LIN {X 0,Y 517.01,Z 148.084,A -85,B 0,C 180,E1 -4953.117,E2 -4953.117} C_VEL
LIN {X 0,Y 516.998,Z 148.087,A -85,B 0,C 180,E1 -4956.243,E2 -4956.243} C_VEL
LIN {X 0,Y 516.949,Z 148.093,A -85,B 0,C 180,E1 -4959.389,E2 -4959.389} C_VEL
LIN {X 0,Y 516.95,Z 148.094,A -85,B 0,C 180,E1 -4961.808,E2 -4961.808} C_VEL
LIN {X 0,Y 516.941,Z 148.093,A -85,B 0,C 180,E1 -4965.147,E2 -4965.147} C_VEL
LIN {X 0,Y 516.922,Z 148.096,A -85,B 0,C 180,E1 -4968.222,E2 -4968.222} C_VEL
LIN {X 0,Y 516.909,Z 148.099,A -85,B 0,C 180,E1 -4970.702,E2 -4970.702} C_VEL
LIN {X 0,Y 516.909,Z 148.099,A -85,B 0,C 180,E1 -4974.072,E2 -4974.072} C_VEL
LIN {X 0,Y 516.923,Z 148.097,A -85,B 0,C 180,E1 -4976.658,E2 -4976.658} C_VEL
LIN {X 0,Y 516.909,Z 148.098,A -85,B 0,C 180,E1 -4979.524,E2 -4979.524} C_VEL
LIN {X 0,Y 516.895,Z 148.101,A -85,B 0,C 180,E1 -4982.544,E2 -4982.544} C_VEL
LIN {X 0,Y 516.863,Z 148.104,A -85,B 0,C 180,E1 -4985.33,E2 -4985.33} C_VEL
LIN {X 0,Y 516.878,Z 148.101,A -85,B 0,C 180,E1 -4987.943,E2 -4987.943} C_VEL
LIN {X 0,Y 516.883,Z 148.101,A -85,B 0,C 180,E1 -4990.742,E2 -4990.742} C_VEL
LIN {X 0,Y 516.882,Z 148.101,A -85,B 0,C 180,E1 -4992.832,E2 -4992.832} C_VEL
LIN {X 0,Y 516.921,Z 148.097,A -85,B 0,C 180,E1 -4995.01,E2 -4995.01} C_VEL
LIN {X 0,Y 516.911,Z 148.1,A -85,B 0,C 180,E1 -4998.399,E2 -4998.399} C_VEL
LIN {X 0,Y 516.88,Z 148.101,A -85,B 0,C 180,E1 -5001.285,E2 -5001.285} C_VEL
LIN {X 0,Y 516.885,Z 148.102,A -85,B 0,C 180,E1 -5004.221,E2 -5004.221} C_VEL
LIN {X 0,Y 516.88,Z 148.102,A -85,B 0,C 180,E1 -5007.053,E2 -5007.053} C_VEL
LIN {X 0,Y 516.891,Z 148.098,A -85,B 0,C 180,E1 -5009.797,E2 -5009.797} C_VEL
LIN {X 0,Y 516.925,Z 148.096,A -85,B 0,C 180,E1 -5012.468,E2 -5012.468} C_VEL
LIN {X 0,Y 516.908,Z 148.1,A -85,B 0,C 180,E1 -5015.072,E2 -5015.072} C_VEL
LIN {X 0,Y 516.886,Z 148.101,A -85,B 0,C 180,E1 -5018.463,E2 -5018.463} C_VEL
LIN {X 0,Y 516.901,Z 148.1,A -85,B 0,C 180,E1 -5020.955,E2 -5020.955} C_VEL
LIN {X 0,Y 516.906,Z 148.099,A -85,B 0,C 180,E1 -5023.41,E2 -5023.41} C_VEL
LIN {X 0,Y 516.893,Z 148.1,A -85,B 0,C 180,E1 -5025.834,E2 -5025.834} C_VEL
LIN {X 0,Y 516.967,Z 148.092,A -85,B 0,C 180,E1 -5028.234,E2 -5028.234} C_VEL
LIN {X 0,Y 516.96,Z 148.091,A -85,B 0,C 180,E1 -5031.4,E2 -5031.4} C_VEL
LIN {X 0,Y 517.012,Z 148.085,A -85,B 0,C 180,E1 -5033.757,E2 -5033.757} C_VEL
LIN {X 0,Y 517.086,Z 148.075,A -85,B 0,C 180,E1 -5037.664,E2 -5037.664} C_VEL
LIN {X 0,Y 517.094,Z 148.074,A -85,B 0,C 180,E1 -5040.779,E2 -5040.779} C_VEL
LIN {X 0,Y 517.013,Z 148.086,A -85,B 0,C 180,E1 -5043.117,E2 -5043.117} C_VEL
LIN {X 0,Y 516.996,Z 148.088,A -85,B 0,C 180,E1 -5046.244,E2 -5046.244} C_VEL
LIN {X 0,Y 516.945,Z 148.094,A -85,B 0,C 180,E1 -5049.39,E2 -5049.39} C_VEL
LIN {X 0,Y 516.955,Z 148.093,A -85,B 0,C 180,E1 -5051.807,E2 -5051.807} C_VEL
LIN {X 0,Y 516.946,Z 148.095,A -85,B 0,C 180,E1 -5055.146,E2 -5055.146} C_VEL
LIN {X 0,Y 516.927,Z 148.096,A -85,B 0,C 180,E1 -5058.222,E2 -5058.222} C_VEL
LIN {X 0,Y 516.915,Z 148.097,A -85,B 0,C 180,E1 -5060.702,E2 -5060.702} C_VEL
LIN {X 0,Y 516.904,Z 148.098,A -85,B 0,C 180,E1 -5064.073,E2 -5064.073} C_VEL
LIN {X 0,Y 516.928,Z 148.094,A -85,B 0,C 180,E1 -5066.658,E2 -5066.658} C_VEL
LIN {X 0,Y 516.913,Z 148.1,A -85,B 0,C 180,E1 -5069.524,E2 -5069.524} C_VEL
LIN {X 0,Y 516.897,Z 148.098,A -85,B 0,C 180,E1 -5072.543,E2 -5072.543} C_VEL
LIN {X 0,Y 516.868,Z 148.104,A -85,B 0,C 180,E1 -5075.33,E2 -5075.33} C_VEL
LIN {X 0,Y 516.882,Z 148.104,A -85,B 0,C 180,E1 -5077.943,E2 -5077.943} C_VEL
LIN {X 0,Y 516.885,Z 148.101,A -85,B 0,C 180,E1 -5080.742,E2 -5080.742} C_VEL
LIN {X 0,Y 516.885,Z 148.101,A -85,B 0,C 180,E1 -5082.832,E2 -5082.832} C_VEL
LIN {X 0,Y 516.926,Z 148.095,A -85,B 0,C 180,E1 -5085.01,E2 -5085.01} C_VEL
LIN {X 0,Y 516.916,Z 148.096,A -85,B 0,C 180,E1 -5088.399,E2 -5088.399} C_VEL
LIN {X 0,Y 516.917,Z 148.208,A -85,B 0,C 180,E1 -5091.168,E2 -5091.168} C_VEL
LIN {X 0,Y 518.075,Z 154.921,A -85,B 0,C 180,E1 -5093.836,E2 -5093.836} C_VEL
LIN {X 0,Y 518.083,Z 160.598,A -85,B 0,C 180,E1 -5095.842,E2 -5095.842} C_VEL
LIN {X 0,Y 517.83,Z 169.691,A -85,B 0,C 180,E1 -5098.953,E2 -5098.953} C_VEL
LIN {X 0,Y 517.591,Z 178.692,A -85,B 0,C 180,E1 -5101.957,E2 -5101.957} C_VEL
LIN {X 0,Y 517.294,Z 188.282,A -85,B 0,C 180,E1 -5105.092,E2 -5105.092} C_VEL
LIN {X 0,Y 517.074,Z 197.549,A -85,B 0,C 180,E1 -5108.051,E2 -5108.051} C_VEL
LIN {X 0,Y 516.881,Z 206.816,A -85,B 0,C 180,E1 -5110.954,E2 -5110.954} C_VEL
LIN {X 0,Y 516.684,Z 217.407,A -85,B 0,C 180,E1 -5114.214,E2 -5114.214} C_VEL
LIN {X 0,Y 516.588,Z 223.736,A -85,B 0,C 180,E1 -5116.095,E2 -5116.095} C_VEL
LIN {X 0,Y 518.516,Z 236.185,A -85,B 0,C 180,E1 -5116.429,E2 -5116.429} C_VEL
LIN {X 0,Y 518.261,Z 248.986,A -85,B 0,C 180,E1 -5116.871,E2 -5116.871} C_VEL
LIN {X 0,Y 517.942,Z 261.176,A -85,B 0,C 180,E1 -5117.461,E2 -5117.461} C_VEL
LIN {X 0,Y 517.617,Z 273.589,A -85,B 0,C 180,E1 -5118.249,E2 -5118.249} C_VEL
LIN {X 0,Y 517.327,Z 284.471,A -85,B 0,C 180,E1 -5119.135,E2 -5119.135} C_VEL
LIN {X 0,Y 517.045,Z 293.335,A -85,B 0,C 180,E1 -5120.02,E2 -5120.02} C_VEL
LIN {X 0,Y 516.814,Z 302.961,A -85,B 0,C 180,E1 -5121.2,E2 -5121.2} C_VEL
LIN {X 0,Y 516.563,Z 310.622,A -85,B 0,C 180,E1 -5122.377,E2 -5122.377} C_VEL
LIN {X 0,Y 516.427,Z 317.68,A -85,B 0,C 180,E1 -5123.75,E2 -5123.75} C_VEL
LIN {X 0,Y 516.313,Z 322.373,A -85,B 0,C 180,E1 -5124.924,E2 -5124.924} C_VEL
LIN {X 0,Y 516.355,Z 325.958,A -85,B 0,C 180,E1 -5126.098,E2 -5126.098} C_VEL
LIN {X 0,Y 516.282,Z 327.808,A -85,B 0,C 180,E1 -5126.879,E2 -5126.879} C_VEL
LIN {X 0,Y 516.261,Z 329.197,A -85,B 0,C 180,E1 -5127.66,E2 -5127.66} C_VEL
LIN {X 0,Y 516.16,Z 330.786,A -85,B 0,C 180,E1 -5129.22,E2 -5129.22} C_VEL
LIN {X 0,Y 516.154,Z 331,A -85,B 0,C 180,E1 -5130,E2 -5130} C_VEL
LIN {X 0,Y 516.192,Z 330.185,A -85,B 0,C 180,E1 -5131.561,E2 -5131.561} C_VEL
LIN {X 0,Y 516.262,Z 329.198,A -85,B 0,C 180,E1 -5132.341,E2 -5132.341} C_VEL
LIN {X 0,Y 516.283,Z 327.81,A -85,B 0,C 180,E1 -5133.121,E2 -5133.121} C_VEL
LIN {X 0,Y 516.344,Z 324.895,A -85,B 0,C 180,E1 -5134.293,E2 -5134.293} C_VEL
LIN {X 0,Y 516.406,Z 320.948,A -85,B 0,C 180,E1 -5135.467,E2 -5135.467} C_VEL
LIN {X 0,Y 516.487,Z 315.032,A -85,B 0,C 180,E1 -5136.808,E2 -5136.808} C_VEL
LIN {X 0,Y 516.641,Z 308.236,A -85,B 0,C 180,E1 -5138.015,E2 -5138.015} C_VEL
LIN {X 0,Y 516.868,Z 299.99,A -85,B 0,C 180,E1 -5139.194,E2 -5139.194} C_VEL
LIN {X 0,Y 517.081,Z 291.537,A -85,B 0,C 180,E1 -5140.177,E2 -5140.177} C_VEL
LIN {X 0,Y 517.435,Z 281.094,A -85,B 0,C 180,E1 -5141.16,E2 -5141.16} C_VEL
LIN {X 0,Y 517.698,Z 269.801,A -85,B 0,C 180,E1 -5142.014,E2 -5142.014} C_VEL
LIN {X 0,Y 517.987,Z 259.405,A -85,B 0,C 180,E1 -5142.638,E2 -5142.638} C_VEL
LIN {X 0,Y 518.27,Z 247.759,A -85,B 0,C 180,E1 -5143.179,E2 -5143.179} C_VEL
LIN {X 0,Y 518.431,Z 234.797,A -85,B 0,C 180,E1 -5143.611,E2 -5143.611} C_VEL
LIN {X 0,Y 516.571,Z 223.53,A -85,B 0,C 180,E1 -5143.924,E2 -5143.924} C_VEL
LIN {X 0,Y 516.712,Z 214.759,A -85,B 0,C 180,E1 -5146.597,E2 -5146.597} C_VEL
LIN {X 0,Y 516.907,Z 205.491,A -85,B 0,C 180,E1 -5149.458,E2 -5149.458} C_VEL
LIN {X 0,Y 517.1,Z 195.963,A -85,B 0,C 180,E1 -5152.451,E2 -5152.451} C_VEL
LIN {X 0,Y 517.324,Z 186.957,A -85,B 0,C 180,E1 -5155.337,E2 -5155.337} C_VEL
LIN {X 0,Y 517.604,Z 177.641,A -85,B 0,C 180,E1 -5158.374,E2 -5158.374} C_VEL
LIN {X 0,Y 517.843,Z 168.077,A -85,B 0,C 180,E1 -5161.55,E2 -5161.55} C_VEL
LIN {X 0,Y 518.14,Z 158.783,A -85,B 0,C 180,E1 -5164.728,E2 -5164.728} C_VEL
LIN {X 0,Y 518.062,Z 154.855,A -85,B 0,C 180,E1 -5166.166,E2 -5166.166} C_VEL
LIN {X 0,Y 516.901,Z 148.101,A -85,B 0,C 180,E1 -5168.893,E2 -5168.893} C_VEL
LIN {X 0,Y 516.918,Z 148.099,A -85,B 0,C 180,E1 -5171.775,E2 -5171.775} C_VEL
LIN {X 0,Y 516.927,Z 148.097,A -85,B 0,C 180,E1 -5175.01,E2 -5175.01} C_VEL
LIN {X 0,Y 516.919,Z 148.1,A -85,B 0,C 180,E1 -5178.399,E2 -5178.399} C_VEL
LIN {X 0,Y 516.886,Z 148.104,A -85,B 0,C 180,E1 -5181.284,E2 -5181.284} C_VEL
LIN {X 0,Y 516.876,Z 148.104,A -85,B 0,C 180,E1 -5184.22,E2 -5184.22} C_VEL
LIN {X 0,Y 516.901,Z 148.1,A -85,B 0,C 180,E1 -5187.053,E2 -5187.053} C_VEL
LIN {X 0,Y 516.897,Z 148.1,A -85,B 0,C 180,E1 -5189.796,E2 -5189.796} C_VEL
LIN {X 0,Y 516.933,Z 148.097,A -85,B 0,C 180,E1 -5192.467,E2 -5192.467} C_VEL
LIN {X 0,Y 516.914,Z 148.098,A -85,B 0,C 180,E1 -5195.072,E2 -5195.072} C_VEL
LIN {X 0,Y 516.891,Z 148.103,A -85,B 0,C 180,E1 -5198.462,E2 -5198.462} C_VEL
LIN {X 0,Y 516.905,Z 148.099,A -85,B 0,C 180,E1 -5200.955,E2 -5200.955} C_VEL
LIN {X 0,Y 516.91,Z 148.1,A -85,B 0,C 180,E1 -5203.41,E2 -5203.41} C_VEL
LIN {X 0,Y 516.9,Z 148.1,A -85,B 0,C 180,E1 -5205.833,E2 -5205.833} C_VEL
LIN {X 0,Y 516.971,Z 148.091,A -85,B 0,C 180,E1 -5208.233,E2 -5208.233} C_VEL
LIN {X 0,Y 516.973,Z 148.091,A -85,B 0,C 180,E1 -5211.399,E2 -5211.399} C_VEL
LIN {X 0,Y 517.016,Z 148.086,A -85,B 0,C 180,E1 -5213.757,E2 -5213.757} C_VEL
LIN {X 0,Y 517.089,Z 148.077,A -85,B 0,C 180,E1 -5217.663,E2 -5217.663} C_VEL
LIN {X 0,Y 517.098,Z 148.076,A -85,B 0,C 180,E1 -5220.778,E2 -5220.778} C_VEL
LIN {X 0,Y 517.016,Z 148.086,A -85,B 0,C 180,E1 -5223.117,E2 -5223.117} C_VEL
LIN {X 0,Y 517.013,Z 148.087,A -85,B 0,C 180,E1 -5226.243,E2 -5226.243} C_VEL
LIN {X 0,Y 516.957,Z 148.095,A -85,B 0,C 180,E1 -5228.6,E2 -5228.6} C_VEL
LIN {X 0,Y 516.756,Z 148.122,A -85,B 0,C 180,E1 -5230.976,E2 -5230.976} C_VEL
LIN {X 0,Y 516.707,Z 148.583,A -85,B 0,C 180,E1 -5231.772,E2 -5231.772} C_VEL
LIN {X 0,Y 516.661,Z 152.229,A -85,B 0,C 180,E1 -5235.028,E2 -5235.028} C_VEL
LIN {X 0,Y 516.555,Z 155.792,A -85,B 0,C 180,E1 -5238.235,E2 -5238.235} C_VEL
LIN {X 0,Y 516.478,Z 158.499,A -85,B 0,C 180,E1 -5240.719,E2 -5240.719} C_VEL
LIN {X 0,Y 516.437,Z 161.326,A -85,B 0,C 180,E1 -5243.244,E2 -5243.244} C_VEL
LIN {X 0,Y 516.458,Z 164.474,A -85,B 0,C 180,E1 -5246.086,E2 -5246.086} C_VEL
LIN {X 0,Y 516.396,Z 167.117,A -85,B 0,C 180,E1 -5248.446,E2 -5248.446} C_VEL
LIN {X 0,Y 516.39,Z 170.263,A -85,B 0,C 180,E1 -5251.228,E2 -5251.228} C_VEL
LIN {X 0,Y 518.487,Z 180.258,A -85,B 0,C 180,E1 -5251.542,E2 -5251.542} C_VEL
LIN {X 0,Y 518.265,Z 193.68,A -85,B 0,C 180,E1 -5252.043,E2 -5252.043} C_VEL
LIN {X 0,Y 518.01,Z 205.328,A -85,B 0,C 180,E1 -5252.635,E2 -5252.635} C_VEL
LIN {X 0,Y 517.692,Z 216.31,A -85,B 0,C 180,E1 -5253.354,E2 -5253.354} C_VEL
LIN {X 0,Y 517.434,Z 227.438,A -85,B 0,C 180,E1 -5254.28,E2 -5254.28} C_VEL
LIN {X 0,Y 517.201,Z 236.447,A -85,B 0,C 180,E1 -5255.204,E2 -5255.204} C_VEL
LIN {X 0,Y 516.915,Z 244.489,A -85,B 0,C 180,E1 -5256.204,E2 -5256.204} C_VEL
LIN {X 0,Y 516.718,Z 251.395,A -85,B 0,C 180,E1 -5257.247,E2 -5257.247} C_VEL
LIN {X 0,Y 516.568,Z 258.171,A -85,B 0,C 180,E1 -5258.521,E2 -5258.521} C_VEL
LIN {X 0,Y 516.422,Z 263.336,A -85,B 0,C 180,E1 -5259.763,E2 -5259.763} C_VEL
LIN {X 0,Y 516.356,Z 266.685,A -85,B 0,C 180,E1 -5260.791,E2 -5260.791} C_VEL
LIN {X 0,Y 516.322,Z 269.256,A -85,B 0,C 180,E1 -5261.833,E2 -5261.833} C_VEL
LIN {X 0,Y 516.274,Z 270.923,A -85,B 0,C 180,E1 -5262.775,E2 -5262.775} C_VEL
LIN {X 0,Y 515.597,Z 271.786,A -85,B 0,C 180,E1 -5263.42,E2 -5263.42} C_VEL
LIN {X 0,Y 512.694,Z 272.704,A -85,B 0,C 180,E1 -5264.472,E2 -5264.472} C_VEL
LIN {X 0,Y 510.257,Z 272.904,A -85,B 0,C 180,E1 -5265.322,E2 -5265.322} C_VEL
LIN {X 0,Y 509.229,Z 272.712,A -85,B 0,C 180,E1 -5265.979,E2 -5265.979} C_VEL
LIN {X 0,Y 509.157,Z 272.566,A -85,B 0,C 180,E1 -5266.201,E2 -5266.201} C_VEL
LIN {X 0,Y 509.204,Z 271.165,A -85,B 0,C 180,E1 -5267.445,E2 -5267.445} C_VEL
LIN {X 0,Y 509.249,Z 269.144,A -85,B 0,C 180,E1 -5268.514,E2 -5268.514} C_VEL
LIN {X 0,Y 509.305,Z 266.411,A -85,B 0,C 180,E1 -5269.566,E2 -5269.566} C_VEL
LIN {X 0,Y 509.438,Z 261.886,A -85,B 0,C 180,E1 -5270.865,E2 -5270.865} C_VEL
LIN {X 0,Y 509.574,Z 255.616,A -85,B 0,C 180,E1 -5272.237,E2 -5272.237} C_VEL
LIN {X 0,Y 509.751,Z 249.046,A -85,B 0,C 180,E1 -5273.374,E2 -5273.374} C_VEL
LIN {X 0,Y 509.996,Z 241.844,A -85,B 0,C 180,E1 -5274.394,E2 -5274.394} C_VEL
LIN {X 0,Y 510.322,Z 232.216,A -85,B 0,C 180,E1 -5275.503,E2 -5275.503} C_VEL
LIN {X 0,Y 510.604,Z 221.763,A -85,B 0,C 180,E1 -5276.476,E2 -5276.476} C_VEL
LIN {X 0,Y 510.87,Z 210.775,A -85,B 0,C 180,E1 -5277.294,E2 -5277.294} C_VEL
LIN {X 0,Y 511.199,Z 198.854,A -85,B 0,C 180,E1 -5277.984,E2 -5277.984} C_VEL
LIN {X 0,Y 511.527,Z 186.379,A -85,B 0,C 180,E1 -5278.527,E2 -5278.527} C_VEL
LIN {X 0,Y 511.357,Z 179.734,A -85,B 0,C 180,E1 -5278.758,E2 -5278.758} C_VEL
LIN {X 0,Y 509.272,Z 170.174,A -85,B 0,C 180,E1 -5279.07,E2 -5279.07} C_VEL
LIN {X 0,Y 509.287,Z 166.728,A -85,B 0,C 180,E1 -5282.027,E2 -5282.027} C_VEL
LIN {X 0,Y 509.343,Z 163.681,A -85,B 0,C 180,E1 -5284.675,E2 -5284.675} C_VEL
LIN {X 0,Y 509.318,Z 160.344,A -85,B 0,C 180,E1 -5287.595,E2 -5287.595} C_VEL
LIN {X 0,Y 509.349,Z 156.878,A -85,B 0,C 180,E1 -5290.661,E2 -5290.661} C_VEL
LIN {X 0,Y 509.419,Z 154.049,A -85,B 0,C 180,E1 -5293.159,E2 -5293.159} C_VEL
LIN {X 0,Y 509.504,Z 151.26,A -85,B 0,C 180,E1 -5295.624,E2 -5295.624} C_VEL
LIN {X 0,Y 509.523,Z 149.455,A -85,B 0,C 180,E1 -5297.25,E2 -5297.25} C_VEL
LIN {X 0,Y 509.655,Z 149.004,A -85,B 0,C 180,E1 -5298.255,E2 -5298.255} C_VEL
LIN {X 0,Y 509.894,Z 148.972,A -85,B 0,C 180,E1 -5301.279,E2 -5301.279} C_VEL
LIN {X 0,Y 509.941,Z 148.966,A -85,B 0,C 180,E1 -5303.67,E2 -5303.67} C_VEL
LIN {X 0,Y 509.952,Z 148.963,A -85,B 0,C 180,E1 -5306.84,E2 -5306.84} C_VEL
LIN {X 0,Y 510.06,Z 148.95,A -85,B 0,C 180,E1 -5309.21,E2 -5309.21} C_VEL
LIN {X 0,Y 510.053,Z 148.953,A -85,B 0,C 180,E1 -5312.369,E2 -5312.369} C_VEL
LIN {X 0,Y 509.976,Z 148.961,A -85,B 0,C 180,E1 -5315.536,E2 -5315.536} C_VEL
LIN {X 0,Y 509.948,Z 148.965,A -85,B 0,C 180,E1 -5317.921,E2 -5317.921} C_VEL
LIN {X 0,Y 509.91,Z 148.97,A -85,B 0,C 180,E1 -5321.125,E2 -5321.125} C_VEL
LIN {X 0,Y 509.861,Z 148.977,A -85,B 0,C 180,E1 -5324.366,E2 -5324.366} C_VEL
LIN {X 0,Y 509.899,Z 148.972,A -85,B 0,C 180,E1 -5327.652,E2 -5327.652} C_VEL
LIN {X 0,Y 509.883,Z 148.974,A -85,B 0,C 180,E1 -5330.402,E2 -5330.402} C_VEL
LIN {X 0,Y 509.834,Z 148.979,A -85,B 0,C 180,E1 -5333.563,E2 -5333.563} C_VEL
LIN {X 0,Y 509.909,Z 148.971,A -85,B 0,C 180,E1 -5336.379,E2 -5336.379} C_VEL
LIN {X 0,Y 509.874,Z 148.975,A -85,B 0,C 180,E1 -5338.844,E2 -5338.844} C_VEL
LIN {X 0,Y 509.819,Z 148.982,A -85,B 0,C 180,E1 -5341.59,E2 -5341.59} C_VEL
LIN {X 0,Y 509.844,Z 148.976,A -85,B 0,C 180,E1 -5344.414,E2 -5344.414} C_VEL
LIN {X 0,Y 509.814,Z 148.984,A -85,B 0,C 180,E1 -5347.341,E2 -5347.341} C_VEL
LIN {X 0,Y 509.836,Z 148.978,A -85,B 0,C 180,E1 -5350.382,E2 -5350.382} C_VEL
LIN {X 0,Y 509.822,Z 148.981,A -85,B 0,C 180,E1 -5353.063,E2 -5353.063} C_VEL
LIN {X 0,Y 509.829,Z 148.981,A -85,B 0,C 180,E1 -5355.793,E2 -5355.793} C_VEL
LIN {X 0,Y 509.853,Z 148.978,A -85,B 0,C 180,E1 -5358.575,E2 -5358.575} C_VEL
LIN {X 0,Y 509.85,Z 148.978,A -85,B 0,C 180,E1 -5361.787,E2 -5361.787} C_VEL
LIN {X 0,Y 509.841,Z 148.979,A -85,B 0,C 180,E1 -5364.623,E2 -5364.623} C_VEL
LIN {X 0,Y 509.859,Z 148.976,A -85,B 0,C 180,E1 -5367.481,E2 -5367.481} C_VEL
LIN {X 0,Y 509.857,Z 148.977,A -85,B 0,C 180,E1 -5370.274,E2 -5370.274} C_VEL
LIN {X 0,Y 509.883,Z 148.974,A -85,B 0,C 180,E1 -5372.945,E2 -5372.945} C_VEL
LIN {X 0,Y 509.864,Z 148.974,A -85,B 0,C 180,E1 -5375.574,E2 -5375.574} C_VEL
LIN {X 0,Y 509.851,Z 148.977,A -85,B 0,C 180,E1 -5378.999,E2 -5378.999} C_VEL
LIN {X 0,Y 509.862,Z 148.976,A -85,B 0,C 180,E1 -5381.517,E2 -5381.517} C_VEL
LIN {X 0,Y 509.911,Z 148.971,A -85,B 0,C 180,E1 -5384.819,E2 -5384.819} C_VEL
LIN {X 0,Y 509.902,Z 148.971,A -85,B 0,C 180,E1 -5388.124,E2 -5388.124} C_VEL
LIN {X 0,Y 509.908,Z 148.969,A -85,B 0,C 180,E1 -5391.28,E2 -5391.28} C_VEL
LIN {X 0,Y 509.981,Z 148.961,A -85,B 0,C 180,E1 -5393.671,E2 -5393.671} C_VEL
LIN {X 0,Y 510.057,Z 148.951,A -85,B 0,C 180,E1 -5397.631,E2 -5397.631} C_VEL
LIN {X 0,Y 510.065,Z 148.95,A -85,B 0,C 180,E1 -5400.79,E2 -5400.79} C_VEL
LIN {X 0,Y 509.955,Z 148.965,A -85,B 0,C 180,E1 -5403.161,E2 -5403.161} C_VEL
LIN {X 0,Y 509.944,Z 148.967,A -85,B 0,C 180,E1 -5406.33,E2 -5406.33} C_VEL
LIN {X 0,Y 509.906,Z 148.971,A -85,B 0,C 180,E1 -5408.721,E2 -5408.721} C_VEL
LIN {X 0,Y 509.907,Z 148.97,A -85,B 0,C 180,E1 -5411.932,E2 -5411.932} C_VEL
LIN {X 0,Y 509.897,Z 148.973,A -85,B 0,C 180,E1 -5415.242,E2 -5415.242} C_VEL
LIN {X 0,Y 509.885,Z 148.973,A -85,B 0,C 180,E1 -5417.999,E2 -5417.999} C_VEL
LIN {X 0,Y 509.853,Z 148.978,A -85,B 0,C 180,E1 -5421.002,E2 -5421.002} C_VEL
LIN {X 0,Y 509.866,Z 148.976,A -85,B 0,C 180,E1 -5424.427,E2 -5424.427} C_VEL
LIN {X 0,Y 509.887,Z 148.974,A -85,B 0,C 180,E1 -5427.056,E2 -5427.056} C_VEL
LIN {X 0,Y 509.86,Z 148.976,A -85,B 0,C 180,E1 -5429.751,E2 -5429.751} C_VEL
LIN {X 0,Y 509.869,Z 148.974,A -85,B 0,C 180,E1 -5432.773,E2 -5432.773} C_VEL
LIN {X 0,Y 509.828,Z 148.981,A -85,B 0,C 180,E1 -5435.579,E2 -5435.579} C_VEL
LIN {X 0,Y 509.852,Z 148.977,A -85,B 0,C 180,E1 -5438.338,E2 -5438.338} C_VEL
LIN {X 0,Y 509.858,Z 148.978,A -85,B 0,C 180,E1 -5441.426,E2 -5441.426} C_VEL
LIN {X 0,Y 509.859,Z 148.973,A -85,B 0,C 180,E1 -5444.668,E2 -5444.668} C_VEL
LIN {X 0,Y 509.858,Z 148.975,A -85,B 0,C 180,E1 -5448.104,E2 -5448.104} C_VEL
LIN {X 0,Y 509.876,Z 149.163,A -85,B 0,C 180,E1 -5450.905,E2 -5450.905} C_VEL
LIN {X 0,Y 511.095,Z 156.154,A -85,B 0,C 180,E1 -5453.752,E2 -5453.752} C_VEL
LIN {X 0,Y 511.114,Z 161.509,A -85,B 0,C 180,E1 -5455.683,E2 -5455.683} C_VEL
LIN {X 0,Y 510.88,Z 169.695,A -85,B 0,C 180,E1 -5458.53,E2 -5458.53} C_VEL
LIN {X 0,Y 510.591,Z 179.233,A -85,B 0,C 180,E1 -5461.755,E2 -5461.755} C_VEL
LIN {X 0,Y 510.302,Z 188.282,A -85,B 0,C 180,E1 -5464.727,E2 -5464.727} C_VEL
LIN {X 0,Y 510.081,Z 197.673,A -85,B 0,C 180,E1 -5467.774,E2 -5467.774} C_VEL
LIN {X 0,Y 509.859,Z 206.816,A -85,B 0,C 180,E1 -5470.681,E2 -5470.681} C_VEL
LIN {X 0,Y 509.647,Z 217.407,A -85,B 0,C 180,E1 -5473.99,E2 -5473.99} C_VEL
LIN {X 0,Y 509.54,Z 223.736,A -85,B 0,C 180,E1 -5475.899,E2 -5475.899} C_VEL
LIN {X 0,Y 511.617,Z 236.642,A -85,B 0,C 180,E1 -5476.255,E2 -5476.255} C_VEL
LIN {X 0,Y 511.36,Z 248.985,A -85,B 0,C 180,E1 -5476.691,E2 -5476.691} C_VEL
LIN {X 0,Y 510.995,Z 261.176,A -85,B 0,C 180,E1 -5477.288,E2 -5477.288} C_VEL
LIN {X 0,Y 510.742,Z 271.848,A -85,B 0,C 180,E1 -5477.964,E2 -5477.964} C_VEL
LIN {X 0,Y 510.416,Z 282.264,A -85,B 0,C 180,E1 -5478.785,E2 -5478.785} C_VEL
LIN {X 0,Y 510.07,Z 291.54,A -85,B 0,C 180,E1 -5479.682,E2 -5479.682} C_VEL
LIN {X 0,Y 509.846,Z 299.992,A -85,B 0,C 180,E1 -5480.679,E2 -5480.679} C_VEL
LIN {X 0,Y 509.585,Z 308.237,A -85,B 0,C 180,E1 -5481.873,E2 -5481.873} C_VEL
LIN {X 0,Y 509.419,Z 314.878,A -85,B 0,C 180,E1 -5483.067,E2 -5483.067} C_VEL
LIN {X 0,Y 509.344,Z 320.95,A -85,B 0,C 180,E1 -5484.457,E2 -5484.457} C_VEL
LIN {X 0,Y 509.234,Z 324.895,A -85,B 0,C 180,E1 -5485.647,E2 -5485.647} C_VEL
LIN {X 0,Y 509.201,Z 327.808,A -85,B 0,C 180,E1 -5486.835,E2 -5486.835} C_VEL
LIN {X 0,Y 509.162,Z 329.196,A -85,B 0,C 180,E1 -5487.627,E2 -5487.627} C_VEL
LIN {X 0,Y 509.073,Z 330.786,A -85,B 0,C 180,E1 -5489.209,E2 -5489.209} C_VEL
LIN {X 0,Y 509.065,Z 331,A -85,B 0,C 180,E1 -5490,E2 -5490} C_VEL
LIN {X 0,Y 509.113,Z 330.185,A -85,B 0,C 180,E1 -5491.582,E2 -5491.582} C_VEL
LIN {X 0,Y 509.162,Z 329.198,A -85,B 0,C 180,E1 -5492.373,E2 -5492.373} C_VEL
LIN {X 0,Y 509.201,Z 327.81,A -85,B 0,C 180,E1 -5493.165,E2 -5493.165} C_VEL
LIN {X 0,Y 509.234,Z 324.895,A -85,B 0,C 180,E1 -5494.353,E2 -5494.353} C_VEL
LIN {X 0,Y 509.345,Z 320.948,A -85,B 0,C 180,E1 -5495.543,E2 -5495.543} C_VEL
LIN {X 0,Y 509.411,Z 315.281,A -85,B 0,C 180,E1 -5496.854,E2 -5496.854} C_VEL
LIN {X 0,Y 509.586,Z 308.235,A -85,B 0,C 180,E1 -5498.127,E2 -5498.127} C_VEL
LIN {X 0,Y 509.847,Z 299.99,A -85,B 0,C 180,E1 -5499.321,E2 -5499.321} C_VEL
LIN {X 0,Y 510.07,Z 291.537,A -85,B 0,C 180,E1 -5500.319,E2 -5500.319} C_VEL
LIN {X 0,Y 510.452,Z 281.093,A -85,B 0,C 180,E1 -5501.315,E2 -5501.315} C_VEL
LIN {X 0,Y 510.731,Z 270.53,A -85,B 0,C 180,E1 -5502.129,E2 -5502.129} C_VEL
LIN {X 0,Y 511.044,Z 259.404,A -85,B 0,C 180,E1 -5502.812,E2 -5502.812} C_VEL
LIN {X 0,Y 511.376,Z 247.759,A -85,B 0,C 180,E1 -5503.36,E2 -5503.36} C_VEL
LIN {X 0,Y 511.433,Z 235.254,A -85,B 0,C 180,E1 -5503.788,E2 -5503.788} C_VEL
LIN {X 0,Y 509.531,Z 223.53,A -85,B 0,C 180,E1 -5504.121,E2 -5504.121} C_VEL
LIN {X 0,Y 509.718,Z 213.435,A -85,B 0,C 180,E1 -5507.244,E2 -5507.244} C_VEL
LIN {X 0,Y 509.925,Z 204.167,A -85,B 0,C 180,E1 -5510.155,E2 -5510.155} C_VEL
LIN {X 0,Y 510.123,Z 194.9,A -85,B 0,C 180,E1 -5513.12,E2 -5513.12} C_VEL
LIN {X 0,Y 510.372,Z 185.572,A -85,B 0,C 180,E1 -5516.146,E2 -5516.146} C_VEL
LIN {X 0,Y 510.608,Z 177.504,A -85,B 0,C 180,E1 -5518.799,E2 -5518.799} C_VEL
LIN {X 0,Y 510.855,Z 169.425,A -85,B 0,C 180,E1 -5521.519,E2 -5521.519} C_VEL
LIN {X 0,Y 511.178,Z 159.957,A -85,B 0,C 180,E1 -5524.793,E2 -5524.793} C_VEL
LIN {X 0,Y 510.964,Z 155.063,A -85,B 0,C 180,E1 -5526.65,E2 -5526.65} C_VEL
LIN {X 0,Y 509.852,Z 148.979,A -85,B 0,C 180,E1 -5529.225,E2 -5529.225} C_VEL
LIN {X 0,Y 509.862,Z 148.977,A -85,B 0,C 180,E1 -5531.897,E2 -5531.897} C_VEL
LIN {X 0,Y 509.861,Z 148.979,A -85,B 0,C 180,E1 -5535.332,E2 -5535.332} C_VEL
LIN {X 0,Y 509.861,Z 148.979,A -85,B 0,C 180,E1 -5538.575,E2 -5538.575} C_VEL
LIN {X 0,Y 509.856,Z 148.979,A -85,B 0,C 180,E1 -5541.786,E2 -5541.786} C_VEL
LIN {X 0,Y 509.835,Z 148.981,A -85,B 0,C 180,E1 -5544.622,E2 -5544.622} C_VEL
LIN {X 0,Y 509.868,Z 148.976,A -85,B 0,C 180,E1 -5547.481,E2 -5547.481} C_VEL
LIN {X 0,Y 509.863,Z 148.978,A -85,B 0,C 180,E1 -5550.274,E2 -5550.274} C_VEL
LIN {X 0,Y 509.89,Z 148.972,A -85,B 0,C 180,E1 -5552.944,E2 -5552.944} C_VEL
LIN {X 0,Y 509.869,Z 148.976,A -85,B 0,C 180,E1 -5555.574,E2 -5555.574} C_VEL
LIN {X 0,Y 509.855,Z 148.977,A -85,B 0,C 180,E1 -5558.998,E2 -5558.998} C_VEL
LIN {X 0,Y 509.866,Z 148.976,A -85,B 0,C 180,E1 -5561.516,E2 -5561.516} C_VEL
LIN {X 0,Y 509.916,Z 148.97,A -85,B 0,C 180,E1 -5564.819,E2 -5564.819} C_VEL
LIN {X 0,Y 509.906,Z 148.971,A -85,B 0,C 180,E1 -5568.124,E2 -5568.124} C_VEL
LIN {X 0,Y 509.92,Z 148.97,A -85,B 0,C 180,E1 -5571.279,E2 -5571.279} C_VEL
LIN {X 0,Y 509.984,Z 148.963,A -85,B 0,C 180,E1 -5573.67,E2 -5573.67} C_VEL
LIN {X 0,Y 510.06,Z 148.953,A -85,B 0,C 180,E1 -5577.631,E2 -5577.631} C_VEL
LIN {X 0,Y 510.068,Z 148.951,A -85,B 0,C 180,E1 -5580.789,E2 -5580.789} C_VEL
LIN {X 0,Y 509.958,Z 148.965,A -85,B 0,C 180,E1 -5583.16,E2 -5583.16} C_VEL
LIN {X 0,Y 509.982,Z 148.963,A -85,B 0,C 180,E1 -5586.329,E2 -5586.329} C_VEL
LIN {X 0,Y 509.899,Z 148.974,A -85,B 0,C 180,E1 -5588.72,E2 -5588.72} C_VEL
LIN {X 0,Y 509.695,Z 149.001,A -85,B 0,C 180,E1 -5591.13,E2 -5591.13} C_VEL
LIN {X 0,Y 509.635,Z 149.582,A -85,B 0,C 180,E1 -5591.938,E2 -5591.938} C_VEL
LIN {X 0,Y 509.589,Z 153.184,A -85,B 0,C 180,E1 -5595.191,E2 -5595.191} C_VEL
LIN {X 0,Y 509.479,Z 156.8,A -85,B 0,C 180,E1 -5598.498,E2 -5598.498} C_VEL
LIN {X 0,Y 509.401,Z 159.606,A -85,B 0,C 180,E1 -5601.021,E2 -5601.021} C_VEL
LIN {X 0,Y 509.348,Z 162.415,A -85,B 0,C 180,E1 -5603.587,E2 -5603.587} C_VEL
LIN {X 0,Y 509.406,Z 165.381,A -85,B 0,C 180,E1 -5606.263,E2 -5606.263} C_VEL
LIN {X 0,Y 509.323,Z 168.295,A -85,B 0,C 180,E1 -5608.878,E2 -5608.878} C_VEL
LIN {X 0,Y 509.335,Z 170.743,A -85,B 0,C 180,E1 -5611.037,E2 -5611.037} C_VEL
LIN {X 0,Y 511.622,Z 181.465,A -85,B 0,C 180,E1 -5611.386,E2 -5611.386} C_VEL
LIN {X 0,Y 511.352,Z 194.845,A -85,B 0,C 180,E1 -5611.901,E2 -5611.901} C_VEL
LIN {X 0,Y 511.06,Z 206.685,A -85,B 0,C 180,E1 -5612.521,E2 -5612.521} C_VEL
LIN {X 0,Y 510.734,Z 217.646,A -85,B 0,C 180,E1 -5613.266,E2 -5613.266} C_VEL
LIN {X 0,Y 510.434,Z 228.789,A -85,B 0,C 180,E1 -5614.221,E2 -5614.221} C_VEL
LIN {X 0,Y 510.153,Z 238.29,A -85,B 0,C 180,E1 -5615.231,E2 -5615.231} C_VEL
LIN {X 0,Y 509.838,Z 246.793,A -85,B 0,C 180,E1 -5616.351,E2 -5616.351} C_VEL
LIN {X 0,Y 509.639,Z 254.187,A -85,B 0,C 180,E1 -5617.558,E2 -5617.558} C_VEL
LIN {X 0,Y 509.46,Z 260.61,A -85,B 0,C 180,E1 -5618.878,E2 -5618.878} C_VEL
LIN {X 0,Y 509.355,Z 264.546,A -85,B 0,C 180,E1 -5619.91,E2 -5619.91} C_VEL
LIN {X 0,Y 509.266,Z 267.894,A -85,B 0,C 180,E1 -5621.025,E2 -5621.025} C_VEL
LIN {X 0,Y 509.256,Z 269.76,A -85,B 0,C 180,E1 -5621.821,E2 -5621.821} C_VEL
LIN {X 0,Y 509.196,Z 271.693,A -85,B 0,C 180,E1 -5622.986,E2 -5622.986} C_VEL
LIN {X 0,Y 509.15,Z 272.744,A -85,B 0,C 180,E1 -5624.128,E2 -5624.128} C_VEL
LIN {X 0,Y 509.147,Z 272.987,A -85,B 0,C 180,E1 -5625.253,E2 -5625.253} C_VEL
LIN {X 0,Y 509.157,Z 272.566,A -85,B 0,C 180,E1 -5626.201,E2 -5626.201} C_VEL
LIN {X 0,Y 508.521,Z 272.042,A -85,B 0,C 180,E1 -5626.861,E2 -5626.861} C_VEL
LIN {X 0,Y 505.692,Z 270.711,A -85,B 0,C 180,E1 -5627.926,E2 -5627.926} C_VEL
LIN {X 0,Y 503.304,Z 269.091,A -85,B 0,C 180,E1 -5628.771,E2 -5628.771} C_VEL
LIN {X 0,Y 502.299,Z 267.463,A -85,B 0,C 180,E1 -5629.412,E2 -5629.412} C_VEL
LIN {X 0,Y 502.23,Z 266.832,A -85,B 0,C 180,E1 -5629.626,E2 -5629.626} C_VEL
LIN {X 0,Y 502.383,Z 262.138,A -85,B 0,C 180,E1 -5630.985,E2 -5630.985} C_VEL
LIN {X 0,Y 502.51,Z 256.492,A -85,B 0,C 180,E1 -5632.242,E2 -5632.242} C_VEL
LIN {X 0,Y 502.755,Z 249.052,A -85,B 0,C 180,E1 -5633.551,E2 -5633.551} C_VEL
LIN {X 0,Y 503.058,Z 240.93,A -85,B 0,C 180,E1 -5634.687,E2 -5634.687} C_VEL
LIN {X 0,Y 503.336,Z 232.635,A -85,B 0,C 180,E1 -5635.644,E2 -5635.644} C_VEL
LIN {X 0,Y 503.643,Z 222.563,A -85,B 0,C 180,E1 -5636.597,E2 -5636.597} C_VEL
LIN {X 0,Y 503.916,Z 212.012,A -85,B 0,C 180,E1 -5637.405,E2 -5637.405} C_VEL
LIN {X 0,Y 504.277,Z 200.675,A -85,B 0,C 180,E1 -5638.087,E2 -5638.087} C_VEL
LIN {X 0,Y 504.63,Z 187.628,A -85,B 0,C 180,E1 -5638.677,E2 -5638.677} C_VEL
LIN {X 0,Y 504.575,Z 181.35,A -85,B 0,C 180,E1 -5638.902,E2 -5638.902} C_VEL
LIN {X 0,Y 502.172,Z 170.533,A -85,B 0,C 180,E1 -5639.281,E2 -5639.281} C_VEL
LIN {X 0,Y 502.206,Z 166.815,A -85,B 0,C 180,E1 -5642.496,E2 -5642.496} C_VEL
LIN {X 0,Y 502.237,Z 163.737,A -85,B 0,C 180,E1 -5645.178,E2 -5645.178} C_VEL
LIN {X 0,Y 502.27,Z 160.751,A -85,B 0,C 180,E1 -5647.802,E2 -5647.802} C_VEL
LIN {X 0,Y 502.281,Z 157.844,A -85,B 0,C 180,E1 -5650.378,E2 -5650.378} C_VEL
LIN {X 0,Y 502.363,Z 154.991,A -85,B 0,C 180,E1 -5652.915,E2 -5652.915} C_VEL
LIN {X 0,Y 502.439,Z 152.19,A -85,B 0,C 180,E1 -5655.417,E2 -5655.417} C_VEL
LIN {X 0,Y 502.447,Z 150.358,A -85,B 0,C 180,E1 -5657.067,E2 -5657.067} C_VEL
LIN {X 0,Y 502.597,Z 149.883,A -85,B 0,C 180,E1 -5658.189,E2 -5658.189} C_VEL
LIN {X 0,Y 502.848,Z 149.849,A -85,B 0,C 180,E1 -5661.156,E2 -5661.156} C_VEL
LIN {X 0,Y 502.893,Z 149.843,A -85,B 0,C 180,E1 -5663.581,E2 -5663.581} C_VEL
LIN {X 0,Y 502.895,Z 149.842,A -85,B 0,C 180,E1 -5666.795,E2 -5666.795} C_VEL
LIN {X 0,Y 503.031,Z 149.826,A -85,B 0,C 180,E1 -5669.199,E2 -5669.199} C_VEL
LIN {X 0,Y 502.901,Z 149.843,A -85,B 0,C 180,E1 -5671.601,E2 -5671.601} C_VEL
LIN {X 0,Y 502.895,Z 149.842,A -85,B 0,C 180,E1 -5673.204,E2 -5673.204} C_VEL
LIN {X 0,Y 502.902,Z 149.842,A -85,B 0,C 180,E1 -5676.419,E2 -5676.419} C_VEL
LIN {X 0,Y 502.87,Z 149.846,A -85,B 0,C 180,E1 -5678.843,E2 -5678.843} C_VEL
LIN {X 0,Y 502.843,Z 149.851,A -85,B 0,C 180,E1 -5682.102,E2 -5682.102} C_VEL
LIN {X 0,Y 502.845,Z 149.85,A -85,B 0,C 180,E1 -5685.4,E2 -5685.4} C_VEL
LIN {X 0,Y 502.843,Z 149.851,A -85,B 0,C 180,E1 -5688.122,E2 -5688.122} C_VEL
LIN {X 0,Y 502.825,Z 149.853,A -85,B 0,C 180,E1 -5690.536,E2 -5690.536} C_VEL
LIN {X 0,Y 502.794,Z 149.858,A -85,B 0,C 180,E1 -5693.04,E2 -5693.04} C_VEL
LIN {X 0,Y 502.837,Z 149.851,A -85,B 0,C 180,E1 -5695.676,E2 -5695.676} C_VEL
LIN {X 0,Y 502.837,Z 149.849,A -85,B 0,C 180,E1 -5698.373,E2 -5698.373} C_VEL
LIN {X 0,Y 502.791,Z 149.858,A -85,B 0,C 180,E1 -5701.499,E2 -5701.499} C_VEL
LIN {X 0,Y 502.801,Z 149.855,A -85,B 0,C 180,E1 -5703.994,E2 -5703.994} C_VEL
LIN {X 0,Y 502.775,Z 149.86,A -85,B 0,C 180,E1 -5707.178,E2 -5707.178} C_VEL
LIN {X 0,Y 502.786,Z 149.857,A -85,B 0,C 180,E1 -5710.015,E2 -5710.015} C_VEL
LIN {X 0,Y 502.8,Z 149.856,A -85,B 0,C 180,E1 -5712.2,E2 -5712.2} C_VEL
LIN {X 0,Y 502.799,Z 149.856,A -85,B 0,C 180,E1 -5715.469,E2 -5715.469} C_VEL
LIN {X 0,Y 502.817,Z 149.853,A -85,B 0,C 180,E1 -5718.934,E2 -5718.934} C_VEL
LIN {X 0,Y 502.792,Z 149.857,A -85,B 0,C 180,E1 -5722.047,E2 -5722.047} C_VEL
LIN {X 0,Y 502.802,Z 149.855,A -85,B 0,C 180,E1 -5725.035,E2 -5725.035} C_VEL
LIN {X 0,Y 502.781,Z 149.858,A -85,B 0,C 180,E1 -5727.916,E2 -5727.916} C_VEL
LIN {X 0,Y 502.822,Z 149.853,A -85,B 0,C 180,E1 -5730.713,E2 -5730.713} C_VEL
LIN {X 0,Y 502.862,Z 149.847,A -85,B 0,C 180,E1 -5733.44,E2 -5733.44} C_VEL
LIN {X 0,Y 502.785,Z 149.857,A -85,B 0,C 180,E1 -5736.086,E2 -5736.086} C_VEL
LIN {X 0,Y 502.784,Z 149.86,A -85,B 0,C 180,E1 -5738.689,E2 -5738.689} C_VEL
LIN {X 0,Y 502.827,Z 149.852,A -85,B 0,C 180,E1 -5741.249,E2 -5741.249} C_VEL
LIN {X 0,Y 502.849,Z 149.851,A -85,B 0,C 180,E1 -5744.601,E2 -5744.601} C_VEL
LIN {X 0,Y 502.877,Z 149.846,A -85,B 0,C 180,E1 -5748.04,E2 -5748.04} C_VEL
LIN {X 0,Y 502.869,Z 149.846,A -85,B 0,C 180,E1 -5751.157,E2 -5751.157} C_VEL
LIN {X 0,Y 502.93,Z 149.84,A -85,B 0,C 180,E1 -5753.582,E2 -5753.582} C_VEL
LIN {X 0,Y 502.9,Z 149.844,A -85,B 0,C 180,E1 -5756.796,E2 -5756.796} C_VEL
LIN {X 0,Y 503.036,Z 149.826,A -85,B 0,C 180,E1 -5759.2,E2 -5759.2} C_VEL
LIN {X 0,Y 502.901,Z 149.843,A -85,B 0,C 180,E1 -5761.602,E2 -5761.602} C_VEL
LIN {X 0,Y 502.899,Z 149.844,A -85,B 0,C 180,E1 -5763.205,E2 -5763.205} C_VEL
LIN {X 0,Y 502.893,Z 149.846,A -85,B 0,C 180,E1 -5766.42,E2 -5766.42} C_VEL
LIN {X 0,Y 502.866,Z 149.848,A -85,B 0,C 180,E1 -5768.844,E2 -5768.844} C_VEL
LIN {X 0,Y 502.849,Z 149.85,A -85,B 0,C 180,E1 -5772.102,E2 -5772.102} C_VEL
LIN {X 0,Y 502.851,Z 149.85,A -85,B 0,C 180,E1 -5775.4,E2 -5775.4} C_VEL
LIN {X 0,Y 502.843,Z 149.85,A -85,B 0,C 180,E1 -5778.121,E2 -5778.121} C_VEL
LIN {X 0,Y 502.832,Z 149.85,A -85,B 0,C 180,E1 -5780.536,E2 -5780.536} C_VEL
LIN {X 0,Y 502.793,Z 149.856,A -85,B 0,C 180,E1 -5783.041,E2 -5783.041} C_VEL
LIN {X 0,Y 502.843,Z 149.852,A -85,B 0,C 180,E1 -5785.676,E2 -5785.676} C_VEL
LIN {X 0,Y 502.842,Z 149.851,A -85,B 0,C 180,E1 -5788.373,E2 -5788.373} C_VEL
LIN {X 0,Y 502.795,Z 149.857,A -85,B 0,C 180,E1 -5791.499,E2 -5791.499} C_VEL
LIN {X 0,Y 502.791,Z 149.857,A -85,B 0,C 180,E1 -5793.995,E2 -5793.995} C_VEL
LIN {X 0,Y 502.78,Z 149.858,A -85,B 0,C 180,E1 -5797.178,E2 -5797.178} C_VEL
LIN {X 0,Y 502.79,Z 149.857,A -85,B 0,C 180,E1 -5800.015,E2 -5800.015} C_VEL
LIN {X 0,Y 502.805,Z 149.853,A -85,B 0,C 180,E1 -5802.199,E2 -5802.199} C_VEL
LIN {X 0,Y 502.803,Z 149.853,A -85,B 0,C 180,E1 -5805.468,E2 -5805.468} C_VEL
LIN {X 0,Y 502.822,Z 149.853,A -85,B 0,C 180,E1 -5808.934,E2 -5808.934} C_VEL
LIN {X 0,Y 502.808,Z 149.948,A -85,B 0,C 180,E1 -5810.572,E2 -5810.572} C_VEL
LIN {X 0,Y 503.957,Z 156.175,A -85,B 0,C 180,E1 -5813.154,E2 -5813.154} C_VEL
LIN {X 0,Y 504.253,Z 160.027,A -85,B 0,C 180,E1 -5814.662,E2 -5814.662} C_VEL
LIN {X 0,Y 503.958,Z 168.083,A -85,B 0,C 180,E1 -5817.527,E2 -5817.527} C_VEL
LIN {X 0,Y 503.683,Z 176.159,A -85,B 0,C 180,E1 -5820.323,E2 -5820.323} C_VEL
LIN {X 0,Y 503.442,Z 183.972,A -85,B 0,C 180,E1 -5822.988,E2 -5822.988} C_VEL
LIN {X 0,Y 503.213,Z 192.215,A -85,B 0,C 180,E1 -5825.669,E2 -5825.669} C_VEL
LIN {X 0,Y 502.968,Z 201.521,A -85,B 0,C 180,E1 -5828.697,E2 -5828.697} C_VEL
LIN {X 0,Y 502.716,Z 211.598,A -85,B 0,C 180,E1 -5831.924,E2 -5831.924} C_VEL
LIN {X 0,Y 502.514,Z 221.694,A -85,B 0,C 180,E1 -5835.104,E2 -5835.104} C_VEL
LIN {X 0,Y 502.486,Z 223.582,A -85,B 0,C 180,E1 -5835.693,E2 -5835.693} C_VEL
LIN {X 0,Y 504.672,Z 237.098,A -85,B 0,C 180,E1 -5836.075,E2 -5836.075} C_VEL
LIN {X 0,Y 504.403,Z 250.114,A -85,B 0,C 180,E1 -5836.555,E2 -5836.555} C_VEL
LIN {X 0,Y 504.035,Z 262.527,A -85,B 0,C 180,E1 -5837.188,E2 -5837.188} C_VEL
LIN {X 0,Y 503.696,Z 273.59,A -85,B 0,C 180,E1 -5837.919,E2 -5837.919} C_VEL
LIN {X 0,Y 503.371,Z 284.47,A -85,B 0,C 180,E1 -5838.83,E2 -5838.83} C_VEL
LIN {X 0,Y 503.023,Z 293.335,A -85,B 0,C 180,E1 -5839.739,E2 -5839.739} C_VEL
LIN {X 0,Y 502.705,Z 302.961,A -85,B 0,C 180,E1 -5840.951,E2 -5840.951} C_VEL
LIN {X 0,Y 502.471,Z 310.622,A -85,B 0,C 180,E1 -5842.162,E2 -5842.162} C_VEL
LIN {X 0,Y 502.256,Z 317.68,A -85,B 0,C 180,E1 -5843.573,E2 -5843.573} C_VEL
LIN {X 0,Y 502.186,Z 322.373,A -85,B 0,C 180,E1 -5844.781,E2 -5844.781} C_VEL
LIN {X 0,Y 502.152,Z 325.958,A -85,B 0,C 180,E1 -5845.987,E2 -5845.987} C_VEL
LIN {X 0,Y 502.121,Z 327.808,A -85,B 0,C 180,E1 -5846.791,E2 -5846.791} C_VEL
LIN {X 0,Y 502.066,Z 329.195,A -85,B 0,C 180,E1 -5847.593,E2 -5847.593} C_VEL
LIN {X 0,Y 501.99,Z 330.786,A -85,B 0,C 180,E1 -5849.198,E2 -5849.198} C_VEL
LIN {X 0,Y 501.98,Z 331,A -85,B 0,C 180,E1 -5850,E2 -5850} C_VEL
LIN {X 0,Y 502.036,Z 330.185,A -85,B 0,C 180,E1 -5851.605,E2 -5851.605} C_VEL
LIN {X 0,Y 502.066,Z 329.197,A -85,B 0,C 180,E1 -5852.407,E2 -5852.407} C_VEL
LIN {X 0,Y 502.121,Z 327.81,A -85,B 0,C 180,E1 -5853.21,E2 -5853.21} C_VEL
LIN {X 0,Y 502.128,Z 324.895,A -85,B 0,C 180,E1 -5854.415,E2 -5854.415} C_VEL
LIN {X 0,Y 502.26,Z 320.948,A -85,B 0,C 180,E1 -5855.621,E2 -5855.621} C_VEL
LIN {X 0,Y 502.336,Z 314.976,A -85,B 0,C 180,E1 -5857.012,E2 -5857.012} C_VEL
LIN {X 0,Y 502.543,Z 308.235,A -85,B 0,C 180,E1 -5858.242,E2 -5858.242} C_VEL
LIN {X 0,Y 502.812,Z 299.99,A -85,B 0,C 180,E1 -5859.453,E2 -5859.453} C_VEL
LIN {X 0,Y 503.064,Z 291.538,A -85,B 0,C 180,E1 -5860.464,E2 -5860.464} C_VEL
LIN {X 0,Y 503.481,Z 281.092,A -85,B 0,C 180,E1 -5861.474,E2 -5861.474} C_VEL
LIN {X 0,Y 503.794,Z 269.428,A -85,B 0,C 180,E1 -5862.378,E2 -5862.378} C_VEL
LIN {X 0,Y 504.147,Z 257.486,A -85,B 0,C 180,E1 -5863.093,E2 -5863.093} C_VEL
LIN {X 0,Y 504.544,Z 245.162,A -85,B 0,C 180,E1 -5863.647,E2 -5863.647} C_VEL
LIN {X 0,Y 504.516,Z 236.168,A -85,B 0,C 180,E1 -5863.956,E2 -5863.956} C_VEL
LIN {X 0,Y 502.469,Z 223.53,A -85,B 0,C 180,E1 -5864.324,E2 -5864.324} C_VEL
LIN {X 0,Y 502.664,Z 213.435,A -85,B 0,C 180,E1 -5867.494,E2 -5867.494} C_VEL
LIN {X 0,Y 502.906,Z 203.829,A -85,B 0,C 180,E1 -5870.558,E2 -5870.558} C_VEL
LIN {X 0,Y 503.14,Z 194.9,A -85,B 0,C 180,E1 -5873.459,E2 -5873.459} C_VEL
LIN {X 0,Y 503.396,Z 184.854,A -85,B 0,C 180,E1 -5876.681,E2 -5876.681} C_VEL
LIN {X 0,Y 503.582,Z 177.242,A -85,B 0,C 180,E1 -5879.24,E2 -5879.24} C_VEL
LIN {X 0,Y 503.87,Z 169.157,A -85,B 0,C 180,E1 -5882.007,E2 -5882.007} C_VEL
LIN {X 0,Y 504.217,Z 161.153,A -85,B 0,C 180,E1 -5884.853,E2 -5884.853} C_VEL
LIN {X 0,Y 504.111,Z 157.138,A -85,B 0,C 180,E1 -5886.399,E2 -5886.399} C_VEL
LIN {X 0,Y 502.793,Z 149.858,A -85,B 0,C 180,E1 -5889.478,E2 -5889.478} C_VEL
LIN {X 0,Y 502.807,Z 149.857,A -85,B 0,C 180,E1 -5892.199,E2 -5892.199} C_VEL
LIN {X 0,Y 502.805,Z 149.857,A -85,B 0,C 180,E1 -5895.468,E2 -5895.468} C_VEL
LIN {X 0,Y 502.825,Z 149.856,A -85,B 0,C 180,E1 -5898.934,E2 -5898.934} C_VEL
LIN {X 0,Y 502.798,Z 149.858,A -85,B 0,C 180,E1 -5902.046,E2 -5902.046} C_VEL
LIN {X 0,Y 502.804,Z 149.856,A -85,B 0,C 180,E1 -5905.034,E2 -5905.034} C_VEL
LIN {X 0,Y 502.79,Z 149.857,A -85,B 0,C 180,E1 -5907.915,E2 -5907.915} C_VEL
LIN {X 0,Y 502.829,Z 149.852,A -85,B 0,C 180,E1 -5910.712,E2 -5910.712} C_VEL
LIN {X 0,Y 502.868,Z 149.848,A -85,B 0,C 180,E1 -5913.439,E2 -5913.439} C_VEL
LIN {X 0,Y 502.79,Z 149.857,A -85,B 0,C 180,E1 -5916.086,E2 -5916.086} C_VEL
LIN {X 0,Y 502.788,Z 149.858,A -85,B 0,C 180,E1 -5918.689,E2 -5918.689} C_VEL
LIN {X 0,Y 502.831,Z 149.853,A -85,B 0,C 180,E1 -5921.248,E2 -5921.248} C_VEL
LIN {X 0,Y 502.853,Z 149.85,A -85,B 0,C 180,E1 -5924.6,E2 -5924.6} C_VEL
LIN {X 0,Y 502.881,Z 149.846,A -85,B 0,C 180,E1 -5928.039,E2 -5928.039} C_VEL
LIN {X 0,Y 502.878,Z 149.846,A -85,B 0,C 180,E1 -5931.156,E2 -5931.156} C_VEL
LIN {X 0,Y 502.934,Z 149.841,A -85,B 0,C 180,E1 -5933.581,E2 -5933.581} C_VEL
LIN {X 0,Y 502.902,Z 149.844,A -85,B 0,C 180,E1 -5936.795,E2 -5936.795} C_VEL
LIN {X 0,Y 503.039,Z 149.826,A -85,B 0,C 180,E1 -5939.199,E2 -5939.199} C_VEL
LIN {X 0,Y 502.904,Z 149.844,A -85,B 0,C 180,E1 -5941.601,E2 -5941.601} C_VEL
LIN {X 0,Y 502.901,Z 149.844,A -85,B 0,C 180,E1 -5943.204,E2 -5943.204} C_VEL
LIN {X 0,Y 502.934,Z 149.841,A -85,B 0,C 180,E1 -5946.418,E2 -5946.418} C_VEL
LIN {X 0,Y 502.853,Z 149.851,A -85,B 0,C 180,E1 -5948.843,E2 -5948.843} C_VEL
LIN {X 0,Y 502.623,Z 149.882,A -85,B 0,C 180,E1 -5951.289,E2 -5951.289} C_VEL
LIN {X 0,Y 502.548,Z 153.311,A -85,B 0,C 180,E1 -5954.579,E2 -5954.579} C_VEL
LIN {X 0,Y 502.463,Z 156.968,A -85,B 0,C 180,E1 -5957.921,E2 -5957.921} C_VEL
LIN {X 0,Y 502.337,Z 160.665,A -85,B 0,C 180,E1 -5961.331,E2 -5961.331} C_VEL
LIN {X 0,Y 502.274,Z 163.544,A -85,B 0,C 180,E1 -5963.939,E2 -5963.939} C_VEL
LIN {X 0,Y 502.325,Z 166.459,A -85,B 0,C 180,E1 -5966.596,E2 -5966.596} C_VEL
LIN {X 0,Y 502.256,Z 169.471,A -85,B 0,C 180,E1 -5969.324,E2 -5969.324} C_VEL
LIN {X 0,Y 502.262,Z 171.165,A -85,B 0,C 180,E1 -5970.829,E2 -5970.829} C_VEL
LIN {X 0,Y 504.72,Z 182.552,A -85,B 0,C 180,E1 -5971.221,E2 -5971.221} C_VEL
LIN {X 0,Y 504.449,Z 195.286,A -85,B 0,C 180,E1 -5971.721,E2 -5971.721} C_VEL
LIN {X 0,Y 504.158,Z 206.952,A -85,B 0,C 180,E1 -5972.34,E2 -5972.34} C_VEL
LIN {X 0,Y 503.812,Z 217.843,A -85,B 0,C 180,E1 -5973.086,E2 -5973.086} C_VEL
LIN {X 0,Y 503.491,Z 228.913,A -85,B 0,C 180,E1 -5974.043,E2 -5974.043} C_VEL
LIN {X 0,Y 503.195,Z 238.383,A -85,B 0,C 180,E1 -5975.056,E2 -5975.056} C_VEL
LIN {X 0,Y 502.848,Z 246.964,A -85,B 0,C 180,E1 -5976.192,E2 -5976.192} C_VEL
LIN {X 0,Y 502.603,Z 255.037,A -85,B 0,C 180,E1 -5977.531,E2 -5977.531} C_VEL
LIN {X 0,Y 502.434,Z 260.614,A -85,B 0,C 180,E1 -5978.694,E2 -5978.694} C_VEL
LIN {X 0,Y 502.268,Z 265.734,A -85,B 0,C 180,E1 -5980.064,E2 -5980.064} C_VEL
LIN {X 0,Y 502.183,Z 269.851,A -85,B 0,C 180,E1 -5981.619,E2 -5981.619} C_VEL
LIN {X 0,Y 502.142,Z 270.987,A -85,B 0,C 180,E1 -5982.206,E2 -5982.206} C_VEL
LIN {X 0,Y 502.104,Z 272.525,A -85,B 0,C 180,E1 -5983.302,E2 -5983.302} C_VEL
LIN {X 0,Y 502.072,Z 273.347,A -85,B 0,C 180,E1 -5984.447,E2 -5984.447} C_VEL
LIN {X 0,Y 502.074,Z 273.344,A -85,B 0,C 180,E1 -5985.581,E2 -5985.581} C_VEL
LIN {X 0,Y 502.103,Z 272.561,A -85,B 0,C 180,E1 -5986.706,E2 -5986.706} C_VEL
LIN {X 0,Y 502.14,Z 270.914,A -85,B 0,C 180,E1 -5987.884,E2 -5987.884} C_VEL
LIN {X 0,Y 502.197,Z 268.316,A -85,B 0,C 180,E1 -5989.086,E2 -5989.086} C_VEL
LIN {X 0,Y 502.23,Z 266.832,A -85,B 0,C 180,E1 -5989.626,E2 -5989.626} C_VEL
LIN {X 0,Y 501.606,Z 264.894,A -85,B 0,C 180,E1 -5990.258,E2 -5990.258} C_VEL
LIN {X 0,Y 497.587,Z 259.812,A -85,B 0,C 180,E1 -5991.671,E2 -5991.671} C_VEL
LIN {X 0,Y 495.778,Z 256.272,A -85,B 0,C 180,E1 -5992.463,E2 -5992.463} C_VEL
LIN {X 0,Y 495.553,Z 254.225,A -85,B 0,C 180,E1 -5992.854,E2 -5992.854} C_VEL
LIN {X 0,Y 495.877,Z 245.988,A -85,B 0,C 180,E1 -5994.192,E2 -5994.192} C_VEL
LIN {X 0,Y 496.2,Z 237.334,A -85,B 0,C 180,E1 -5995.311,E2 -5995.311} C_VEL
LIN {X 0,Y 496.539,Z 227.226,A -85,B 0,C 180,E1 -5996.373,E2 -5996.373} C_VEL
LIN {X 0,Y 496.877,Z 216.937,A -85,B 0,C 180,E1 -5997.247,E2 -5997.247} C_VEL
LIN {X 0,Y 497.184,Z 205.624,A -85,B 0,C 180,E1 -5998.009,E2 -5998.009} C_VEL
LIN {X 0,Y 497.636,Z 192.657,A -85,B 0,C 180,E1 -5998.675,E2 -5998.675} C_VEL
LIN {X 0,Y 497.718,Z 182.552,A -85,B 0,C 180,E1 -5999.064,E2 -5999.064} C_VEL
LIN {X 0,Y 495.107,Z 170.907,A -85,B 0,C 180,E1 -5999.489,E2 -5999.489} C_VEL
LIN {X 0,Y 495.147,Z 167.921,A -85,B 0,C 180,E1 -6002.07,E2 -6002.07} C_VEL
LIN {X 0,Y 495.188,Z 164.807,A -85,B 0,C 180,E1 -6004.8,E2 -6004.8} C_VEL
LIN {X 0,Y 495.176,Z 161.781,A -85,B 0,C 180,E1 -6007.467,E2 -6007.467} C_VEL
LIN {X 0,Y 495.203,Z 158.833,A -85,B 0,C 180,E1 -6010.086,E2 -6010.086} C_VEL
LIN {X 0,Y 495.3,Z 155.964,A -85,B 0,C 180,E1 -6012.664,E2 -6012.664} C_VEL
LIN {X 0,Y 495.367,Z 153.126,A -85,B 0,C 180,E1 -6015.204,E2 -6015.204} C_VEL
LIN {X 0,Y 495.38,Z 151.281,A -85,B 0,C 180,E1 -6016.88,E2 -6016.88} C_VEL
LIN {X 0,Y 495.545,Z 150.762,A -85,B 0,C 180,E1 -6018.118,E2 -6018.118} C_VEL
LIN {X 0,Y 495.798,Z 150.727,A -85,B 0,C 180,E1 -6021.029,E2 -6021.029} C_VEL
LIN {X 0,Y 495.846,Z 150.72,A -85,B 0,C 180,E1 -6023.489,E2 -6023.489} C_VEL
LIN {X 0,Y 495.839,Z 150.721,A -85,B 0,C 180,E1 -6026.75,E2 -6026.75} C_VEL
LIN {X 0,Y 496.001,Z 150.702,A -85,B 0,C 180,E1 -6029.188,E2 -6029.188} C_VEL
LIN {X 0,Y 495.87,Z 150.719,A -85,B 0,C 180,E1 -6031.624,E2 -6031.624} C_VEL
LIN {X 0,Y 495.84,Z 150.721,A -85,B 0,C 180,E1 -6033.25,E2 -6033.25} C_VEL
LIN {X 0,Y 495.856,Z 150.719,A -85,B 0,C 180,E1 -6036.511,E2 -6036.511} C_VEL
LIN {X 0,Y 495.839,Z 150.721,A -85,B 0,C 180,E1 -6038.97,E2 -6038.97} C_VEL
LIN {X 0,Y 495.825,Z 150.726,A -85,B 0,C 180,E1 -6042.035,E2 -6042.035} C_VEL
LIN {X 0,Y 495.821,Z 150.725,A -85,B 0,C 180,E1 -6045.452,E2 -6045.452} C_VEL
LIN {X 0,Y 495.804,Z 150.726,A -85,B 0,C 180,E1 -6048.247,E2 -6048.247} C_VEL
LIN {X 0,Y 495.771,Z 150.732,A -85,B 0,C 180,E1 -6050.756,E2 -6050.756} C_VEL
LIN {X 0,Y 495.75,Z 150.734,A -85,B 0,C 180,E1 -6053.387,E2 -6053.387} C_VEL
LIN {X 0,Y 495.788,Z 150.729,A -85,B 0,C 180,E1 -6056.068,E2 -6056.068} C_VEL
LIN {X 0,Y 495.769,Z 150.731,A -85,B 0,C 180,E1 -6058.815,E2 -6058.815} C_VEL
LIN {X 0,Y 495.753,Z 150.733,A -85,B 0,C 180,E1 -6061.726,E2 -6061.726} C_VEL
LIN {X 0,Y 495.766,Z 150.731,A -85,B 0,C 180,E1 -6064.694,E2 -6064.694} C_VEL
LIN {X 0,Y 495.727,Z 150.737,A -85,B 0,C 180,E1 -6067.562,E2 -6067.562} C_VEL
LIN {X 0,Y 495.764,Z 150.732,A -85,B 0,C 180,E1 -6070.7,E2 -6070.7} C_VEL
LIN {X 0,Y 495.732,Z 150.734,A -85,B 0,C 180,E1 -6074.001,E2 -6074.001} C_VEL
LIN {X 0,Y 495.724,Z 150.739,A -85,B 0,C 180,E1 -6077.117,E2 -6077.117} C_VEL
LIN {X 0,Y 495.757,Z 150.731,A -85,B 0,C 180,E1 -6079.953,E2 -6079.953} C_VEL
LIN {X 0,Y 495.729,Z 150.736,A -85,B 0,C 180,E1 -6082.553,E2 -6082.553} C_VEL
LIN {X 0,Y 495.775,Z 150.731,A -85,B 0,C 180,E1 -6085.457,E2 -6085.457} C_VEL
LIN {X 0,Y 495.754,Z 150.733,A -85,B 0,C 180,E1 -6088.364,E2 -6088.364} C_VEL
LIN {X 0,Y 495.786,Z 150.729,A -85,B 0,C 180,E1 -6091.507,E2 -6091.507} C_VEL
LIN {X 0,Y 495.79,Z 150.729,A -85,B 0,C 180,E1 -6093.933,E2 -6093.933} C_VEL
LIN {X 0,Y 495.76,Z 150.732,A -85,B 0,C 180,E1 -6097.14,E2 -6097.14} C_VEL
LIN {X 0,Y 495.772,Z 150.733,A -85,B 0,C 180,E1 -6100.11,E2 -6100.11} C_VEL
LIN {X 0,Y 495.764,Z 150.732,A -85,B 0,C 180,E1 -6102.681,E2 -6102.681} C_VEL
LIN {X 0,Y 495.79,Z 150.727,A -85,B 0,C 180,E1 -6105.218,E2 -6105.218} C_VEL
LIN {X 0,Y 495.853,Z 150.722,A -85,B 0,C 180,E1 -6108.555,E2 -6108.555} C_VEL
LIN {X 0,Y 495.838,Z 150.723,A -85,B 0,C 180,E1 -6111.852,E2 -6111.852} C_VEL
LIN {X 0,Y 495.896,Z 150.717,A -85,B 0,C 180,E1 -6114.307,E2 -6114.307} C_VEL
LIN {X 0,Y 495.995,Z 150.702,A -85,B 0,C 180,E1 -6117.564,E2 -6117.564} C_VEL
LIN {X 0,Y 495.985,Z 150.703,A -85,B 0,C 180,E1 -6120.812,E2 -6120.812} C_VEL
LIN {X 0,Y 495.996,Z 150.703,A -85,B 0,C 180,E1 -6122.437,E2 -6122.437} C_VEL
LIN {X 0,Y 495.887,Z 150.717,A -85,B 0,C 180,E1 -6125.694,E2 -6125.694} C_VEL
LIN {X 0,Y 495.837,Z 150.723,A -85,B 0,C 180,E1 -6128.97,E2 -6128.97} C_VEL
LIN {X 0,Y 495.831,Z 150.724,A -85,B 0,C 180,E1 -6132.035,E2 -6132.035} C_VEL
LIN {X 0,Y 495.826,Z 150.724,A -85,B 0,C 180,E1 -6135.452,E2 -6135.452} C_VEL
LIN {X 0,Y 495.81,Z 150.727,A -85,B 0,C 180,E1 -6138.248,E2 -6138.248} C_VEL
LIN {X 0,Y 495.777,Z 150.729,A -85,B 0,C 180,E1 -6140.757,E2 -6140.757} C_VEL
LIN {X 0,Y 495.75,Z 150.735,A -85,B 0,C 180,E1 -6143.388,E2 -6143.388} C_VEL
LIN {X 0,Y 495.793,Z 150.727,A -85,B 0,C 180,E1 -6146.068,E2 -6146.068} C_VEL
LIN {X 0,Y 495.773,Z 150.73,A -85,B 0,C 180,E1 -6148.815,E2 -6148.815} C_VEL
LIN {X 0,Y 495.758,Z 150.735,A -85,B 0,C 180,E1 -6151.725,E2 -6151.725} C_VEL
LIN {X 0,Y 495.765,Z 150.732,A -85,B 0,C 180,E1 -6154.693,E2 -6154.693} C_VEL
LIN {X 0,Y 495.731,Z 150.737,A -85,B 0,C 180,E1 -6157.562,E2 -6157.562} C_VEL
LIN {X 0,Y 495.769,Z 150.732,A -85,B 0,C 180,E1 -6160.7,E2 -6160.7} C_VEL
LIN {X 0,Y 495.736,Z 150.734,A -85,B 0,C 180,E1 -6164.001,E2 -6164.001} C_VEL
LIN {X 0,Y 495.728,Z 150.734,A -85,B 0,C 180,E1 -6167.117,E2 -6167.117} C_VEL
LIN {X 0,Y 495.767,Z 150.784,A -85,B 0,C 180,E1 -6170.261,E2 -6170.261} C_VEL
LIN {X 0,Y 496.989,Z 157.463,A -85,B 0,C 180,E1 -6173.058,E2 -6173.058} C_VEL
LIN {X 0,Y 497.292,Z 161.278,A -85,B 0,C 180,E1 -6174.589,E2 -6174.589} C_VEL
LIN {X 0,Y 496.978,Z 169.289,A -85,B 0,C 180,E1 -6177.495,E2 -6177.495} C_VEL
LIN {X 0,Y 496.686,Z 177.315,A -85,B 0,C 180,E1 -6180.314,E2 -6180.314} C_VEL
LIN {X 0,Y 496.406,Z 185.366,A -85,B 0,C 180,E1 -6183.119,E2 -6183.119} C_VEL
LIN {X 0,Y 496.121,Z 194.698,A -85,B 0,C 180,E1 -6186.189,E2 -6186.189} C_VEL
LIN {X 0,Y 495.894,Z 204.293,A -85,B 0,C 180,E1 -6189.29,E2 -6189.29} C_VEL
LIN {X 0,Y 495.639,Z 213.436,A -85,B 0,C 180,E1 -6192.25,E2 -6192.25} C_VEL
LIN {X 0,Y 495.415,Z 223.582,A -85,B 0,C 180,E1 -6195.485,E2 -6195.485} C_VEL
LIN {X 0,Y 497.581,Z 236.643,A -85,B 0,C 180,E1 -6195.859,E2 -6195.859} C_VEL
LIN {X 0,Y 497.659,Z 243.876,A -85,B 0,C 180,E1 -6196.109,E2 -6196.109} C_VEL
LIN {X 0,Y 497.301,Z 255.506,A -85,B 0,C 180,E1 -6196.62,E2 -6196.62} C_VEL
LIN {X 0,Y 496.957,Z 266.846,A -85,B 0,C 180,E1 -6197.276,E2 -6197.276} C_VEL
LIN {X 0,Y 496.623,Z 277.487,A -85,B 0,C 180,E1 -6198.055,E2 -6198.055} C_VEL
LIN {X 0,Y 496.238,Z 287.647,A -85,B 0,C 180,E1 -6198.978,E2 -6198.978} C_VEL
LIN {X 0,Y 495.928,Z 296.787,A -85,B 0,C 180,E1 -6200.003,E2 -6200.003} C_VEL
LIN {X 0,Y 495.606,Z 305.689,A -85,B 0,C 180,E1 -6201.232,E2 -6201.232} C_VEL
LIN {X 0,Y 495.316,Z 312.849,A -85,B 0,C 180,E1 -6202.458,E2 -6202.458} C_VEL
LIN {X 0,Y 495.175,Z 318.686,A -85,B 0,C 180,E1 -6203.717,E2 -6203.717} C_VEL
LIN {X 0,Y 495.039,Z 323.677,A -85,B 0,C 180,E1 -6205.114,E2 -6205.114} C_VEL
LIN {X 0,Y 495.049,Z 325.959,A -85,B 0,C 180,E1 -6205.93,E2 -6205.93} C_VEL
LIN {X 0,Y 495.043,Z 327.807,A -85,B 0,C 180,E1 -6206.745,E2 -6206.745} C_VEL
LIN {X 0,Y 494.961,Z 330.183,A -85,B 0,C 180,E1 -6208.373,E2 -6208.373} C_VEL
LIN {X 0,Y 494.898,Z 331,A -85,B 0,C 180,E1 -6210,E2 -6210} C_VEL
LIN {X 0,Y 494.961,Z 330.184,A -85,B 0,C 180,E1 -6211.627,E2 -6211.627} C_VEL
LIN {X 0,Y 495.043,Z 327.81,A -85,B 0,C 180,E1 -6213.256,E2 -6213.256} C_VEL
LIN {X 0,Y 495.029,Z 324.895,A -85,B 0,C 180,E1 -6214.479,E2 -6214.479} C_VEL
LIN {X 0,Y 495.21,Z 319.802,A -85,B 0,C 180,E1 -6215.999,E2 -6215.999} C_VEL
LIN {X 0,Y 495.278,Z 313.868,A -85,B 0,C 180,E1 -6217.337,E2 -6217.337} C_VEL
LIN {X 0,Y 495.558,Z 307.002,A -85,B 0,C 180,E1 -6218.564,E2 -6218.564} C_VEL
LIN {X 0,Y 495.852,Z 298.411,A -85,B 0,C 180,E1 -6219.793,E2 -6219.793} C_VEL
LIN {X 0,Y 496.181,Z 289.597,A -85,B 0,C 180,E1 -6220.817,E2 -6220.817} C_VEL
LIN {X 0,Y 496.631,Z 278.742,A -85,B 0,C 180,E1 -6221.841,E2 -6221.841} C_VEL
LIN {X 0,Y 496.898,Z 268.211,A -85,B 0,C 180,E1 -6222.636,E2 -6222.636} C_VEL
LIN {X 0,Y 497.3,Z 255.496,A -85,B 0,C 180,E1 -6223.381,E2 -6223.381} C_VEL
LIN {X 0,Y 497.66,Z 243.861,A -85,B 0,C 180,E1 -6223.891,E2 -6223.891} C_VEL
LIN {X 0,Y 497.577,Z 236.624,A -85,B 0,C 180,E1 -6224.141,E2 -6224.141} C_VEL
LIN {X 0,Y 495.426,Z 223.53,A -85,B 0,C 180,E1 -6224.532,E2 -6224.532} C_VEL
LIN {X 0,Y 495.639,Z 213.435,A -85,B 0,C 180,E1 -6227.75,E2 -6227.75} C_VEL
LIN {X 0,Y 495.887,Z 204.167,A -85,B 0,C 180,E1 -6230.752,E2 -6230.752} C_VEL
LIN {X 0,Y 496.119,Z 194.639,A -85,B 0,C 180,E1 -6233.812,E2 -6233.812} C_VEL
LIN {X 0,Y 496.346,Z 186.47,A -85,B 0,C 180,E1 -6236.455,E2 -6236.455} C_VEL
LIN {X 0,Y 496.556,Z 178.325,A -85,B 0,C 180,E1 -6239.229,E2 -6239.229} C_VEL
LIN {X 0,Y 496.848,Z 170.546,A -85,B 0,C 180,E1 -6241.928,E2 -6241.928} C_VEL
LIN {X 0,Y 497.265,Z 162.291,A -85,B 0,C 180,E1 -6244.942,E2 -6244.942} C_VEL
LIN {X 0,Y 497.154,Z 158.512,A -85,B 0,C 180,E1 -6246.423,E2 -6246.423} C_VEL
LIN {X 0,Y 496.151,Z 152.858,A -85,B 0,C 180,E1 -6248.823,E2 -6248.823} C_VEL
LIN {X 0,Y 495.766,Z 150.734,A -85,B 0,C 180,E1 -6249.842,E2 -6249.842} C_VEL
LIN {X 0,Y 495.73,Z 150.735,A -85,B 0,C 180,E1 -6252.883,E2 -6252.883} C_VEL
LIN {X 0,Y 495.739,Z 150.737,A -85,B 0,C 180,E1 -6255.999,E2 -6255.999} C_VEL
LIN {X 0,Y 495.771,Z 150.734,A -85,B 0,C 180,E1 -6259.3,E2 -6259.3} C_VEL
LIN {X 0,Y 495.734,Z 150.738,A -85,B 0,C 180,E1 -6262.438,E2 -6262.438} C_VEL
LIN {X 0,Y 495.783,Z 150.73,A -85,B 0,C 180,E1 -6265.457,E2 -6265.457} C_VEL
LIN {X 0,Y 495.761,Z 150.735,A -85,B 0,C 180,E1 -6268.364,E2 -6268.364} C_VEL
LIN {X 0,Y 495.793,Z 150.73,A -85,B 0,C 180,E1 -6271.507,E2 -6271.507} C_VEL
LIN {X 0,Y 495.796,Z 150.728,A -85,B 0,C 180,E1 -6273.932,E2 -6273.932} C_VEL
LIN {X 0,Y 495.765,Z 150.732,A -85,B 0,C 180,E1 -6277.139,E2 -6277.139} C_VEL
LIN {X 0,Y 495.776,Z 150.73,A -85,B 0,C 180,E1 -6280.109,E2 -6280.109} C_VEL
LIN {X 0,Y 495.769,Z 150.733,A -85,B 0,C 180,E1 -6282.68,E2 -6282.68} C_VEL
LIN {X 0,Y 495.795,Z 150.728,A -85,B 0,C 180,E1 -6285.217,E2 -6285.217} C_VEL
LIN {X 0,Y 495.857,Z 150.722,A -85,B 0,C 180,E1 -6288.555,E2 -6288.555} C_VEL
LIN {X 0,Y 495.878,Z 150.719,A -85,B 0,C 180,E1 -6291.852,E2 -6291.852} C_VEL
LIN {X 0,Y 495.9,Z 150.715,A -85,B 0,C 180,E1 -6294.306,E2 -6294.306} C_VEL
LIN {X 0,Y 495.998,Z 150.704,A -85,B 0,C 180,E1 -6297.563,E2 -6297.563} C_VEL
LIN {X 0,Y 496.004,Z 150.703,A -85,B 0,C 180,E1 -6300,E2 -6300} C_VEL
LIN {X 0,Y 495.998,Z 150.704,A -85,B 0,C 180,E1 -6302.436,E2 -6302.436} C_VEL
LIN {X 0,Y 495.899,Z 150.719,A -85,B 0,C 180,E1 -6305.693,E2 -6305.693} C_VEL
LIN {X 0,Y 495.871,Z 150.721,A -85,B 0,C 180,E1 -6308.148,E2 -6308.148} C_VEL
LIN {X 0,Y 495.614,Z 150.755,A -85,B 0,C 180,E1 -6310.623,E2 -6310.623} C_VEL
LIN {X 0,Y 495.55,Z 150.763,A -85,B 0,C 180,E1 -6311.452,E2 -6311.452} C_VEL
LIN {X 0,Y 495.51,Z 154.343,A -85,B 0,C 180,E1 -6314.791,E2 -6314.791} C_VEL
LIN {X 0,Y 495.386,Z 158.006,A -85,B 0,C 180,E1 -6318.186,E2 -6318.186} C_VEL
LIN {X 0,Y 495.292,Z 160.802,A -85,B 0,C 180,E1 -6320.777,E2 -6320.777} C_VEL
LIN {X 0,Y 495.222,Z 163.691,A -85,B 0,C 180,E1 -6323.413,E2 -6323.413} C_VEL
LIN {X 0,Y 495.257,Z 166.623,A -85,B 0,C 180,E1 -6326.098,E2 -6326.098} C_VEL
LIN {X 0,Y 495.207,Z 169.653,A -85,B 0,C 180,E1 -6328.85,E2 -6328.85} C_VEL
LIN {X 0,Y 495.198,Z 171.628,A -85,B 0,C 180,E1 -6330.629,E2 -6330.629} C_VEL
LIN {X 0,Y 497.837,Z 183.457,A -85,B 0,C 180,E1 -6331.045,E2 -6331.045} C_VEL
LIN {X 0,Y 497.55,Z 197.031,A -85,B 0,C 180,E1 -6331.596,E2 -6331.596} C_VEL
LIN {X 0,Y 497.188,Z 209.279,A -85,B 0,C 180,E1 -6332.284,E2 -6332.284} C_VEL
LIN {X 0,Y 496.838,Z 220.498,A -85,B 0,C 180,E1 -6333.098,E2 -6333.098} C_VEL
LIN {X 0,Y 496.521,Z 230.422,A -85,B 0,C 180,E1 -6333.993,E2 -6333.993} C_VEL
LIN {X 0,Y 496.219,Z 238.678,A -85,B 0,C 180,E1 -6334.899,E2 -6334.899} C_VEL
LIN {X 0,Y 495.822,Z 247.641,A -85,B 0,C 180,E1 -6336.104,E2 -6336.104} C_VEL
LIN {X 0,Y 495.573,Z 255.463,A -85,B 0,C 180,E1 -6337.423,E2 -6337.423} C_VEL
LIN {X 0,Y 495.365,Z 261.505,A -85,B 0,C 180,E1 -6338.71,E2 -6338.71} C_VEL
LIN {X 0,Y 495.222,Z 266.104,A -85,B 0,C 180,E1 -6339.973,E2 -6339.973} C_VEL
LIN {X 0,Y 495.113,Z 269.505,A -85,B 0,C 180,E1 -6341.208,E2 -6341.208} C_VEL
LIN {X 0,Y 495.043,Z 271.861,A -85,B 0,C 180,E1 -6342.419,E2 -6342.419} C_VEL
LIN {X 0,Y 494.99,Z 273.595,A -85,B 0,C 180,E1 -6344.083,E2 -6344.083} C_VEL
LIN {X 0,Y 494.977,Z 273.85,A -85,B 0,C 180,E1 -6345.229,E2 -6345.229} C_VEL
LIN {X 0,Y 495.01,Z 273.319,A -85,B 0,C 180,E1 -6346.392,E2 -6346.392} C_VEL
LIN {X 0,Y 495.038,Z 271.917,A -85,B 0,C 180,E1 -6347.581,E2 -6347.581} C_VEL
LIN {X 0,Y 495.125,Z 268.491,A -85,B 0,C 180,E1 -6349.236,E2 -6349.236} C_VEL
LIN {X 0,Y 495.22,Z 265.315,A -85,B 0,C 180,E1 -6350.31,E2 -6350.31} C_VEL
LIN {X 0,Y 495.404,Z 260.197,A -85,B 0,C 180,E1 -6351.636,E2 -6351.636} C_VEL
LIN {X 0,Y 495.553,Z 254.225,A -85,B 0,C 180,E1 -6352.854,E2 -6352.854} C_VEL
LIN {X 0,Y 495.029,Z 251.049,A -85,B 0,C 180,E1 -6353.428,E2 -6353.428} C_VEL
LIN {X 0,Y 492.403,Z 245.619,A -85,B 0,C 180,E1 -6354.343,E2 -6354.343} C_VEL
LIN {X 0,Y 489.803,Z 239.613,A -85,B 0,C 180,E1 -6355.213,E2 -6355.213} C_VEL
LIN {X 0,Y 489.32,Z 235.534,A -85,B 0,C 180,E1 -6355.71,E2 -6355.71} C_VEL
LIN {X 0,Y 489.71,Z 225.241,A -85,B 0,C 180,E1 -6356.751,E2 -6356.751} C_VEL
LIN {X 0,Y 490.054,Z 214.248,A -85,B 0,C 180,E1 -6357.643,E2 -6357.643} C_VEL
LIN {X 0,Y 490.436,Z 202.363,A -85,B 0,C 180,E1 -6358.403,E2 -6358.403} C_VEL
LIN {X 0,Y 490.825,Z 190.548,A -85,B 0,C 180,E1 -6358.97,E2 -6358.97} C_VEL
LIN {X 0,Y 490.764,Z 183.326,A -85,B 0,C 180,E1 -6359.249,E2 -6359.249} C_VEL
LIN {X 0,Y 488.053,Z 171.282,A -85,B 0,C 180,E1 -6359.698,E2 -6359.698} C_VEL
LIN {X 0,Y 488.087,Z 167.995,A -85,B 0,C 180,E1 -6362.563,E2 -6362.563} C_VEL
LIN {X 0,Y 488.113,Z 164.856,A -85,B 0,C 180,E1 -6365.32,E2 -6365.32} C_VEL
LIN {X 0,Y 488.101,Z 161.82,A -85,B 0,C 180,E1 -6368.015,E2 -6368.015} C_VEL
LIN {X 0,Y 488.153,Z 158.861,A -85,B 0,C 180,E1 -6370.662,E2 -6370.662} C_VEL
LIN {X 0,Y 488.238,Z 155.968,A -85,B 0,C 180,E1 -6373.268,E2 -6373.268} C_VEL
LIN {X 0,Y 488.274,Z 153.143,A -85,B 0,C 180,E1 -6375.836,E2 -6375.836} C_VEL
LIN {X 0,Y 488.392,Z 151.652,A -85,B 0,C 180,E1 -6377.534,E2 -6377.534} C_VEL
LIN {X 0,Y 488.662,Z 151.619,A -85,B 0,C 180,E1 -6380.062,E2 -6380.062} C_VEL
LIN {X 0,Y 488.857,Z 151.593,A -85,B 0,C 180,E1 -6382.73,E2 -6382.73} C_VEL
LIN {X 0,Y 488.808,Z 151.598,A -85,B 0,C 180,E1 -6385.051,E2 -6385.051} C_VEL
LIN {X 0,Y 488.959,Z 151.58,A -85,B 0,C 180,E1 -6387.528,E2 -6387.528} C_VEL
LIN {X 0,Y 488.951,Z 151.581,A -85,B 0,C 180,E1 -6390.823,E2 -6390.823} C_VEL
LIN {X 0,Y 488.959,Z 151.58,A -85,B 0,C 180,E1 -6392.471,E2 -6392.471} C_VEL
LIN {X 0,Y 488.844,Z 151.595,A -85,B 0,C 180,E1 -6395.776,E2 -6395.776} C_VEL
LIN {X 0,Y 488.814,Z 151.599,A -85,B 0,C 180,E1 -6398.266,E2 -6398.266} C_VEL
LIN {X 0,Y 488.803,Z 151.599,A -85,B 0,C 180,E1 -6401.612,E2 -6401.612} C_VEL
LIN {X 0,Y 488.759,Z 151.604,A -85,B 0,C 180,E1 -6405,E2 -6405} C_VEL
LIN {X 0,Y 488.752,Z 151.604,A -85,B 0,C 180,E1 -6408.442,E2 -6408.442} C_VEL
LIN {X 0,Y 488.705,Z 151.611,A -85,B 0,C 180,E1 -6411.071,E2 -6411.071} C_VEL
LIN {X 0,Y 488.691,Z 151.614,A -85,B 0,C 180,E1 -6413.745,E2 -6413.745} C_VEL
LIN {X 0,Y 488.789,Z 151.601,A -85,B 0,C 180,E1 -6416.944,E2 -6416.944} C_VEL
LIN {X 0,Y 488.707,Z 151.611,A -85,B 0,C 180,E1 -6420.363,E2 -6420.363} C_VEL
LIN {X 0,Y 488.731,Z 151.609,A -85,B 0,C 180,E1 -6423.484,E2 -6423.484} C_VEL
LIN {X 0,Y 488.679,Z 151.615,A -85,B 0,C 180,E1 -6426.355,E2 -6426.355} C_VEL
LIN {X 0,Y 488.699,Z 151.612,A -85,B 0,C 180,E1 -6429.254,E2 -6429.254} C_VEL
LIN {X 0,Y 488.706,Z 151.611,A -85,B 0,C 180,E1 -6431.6,E2 -6431.6} C_VEL
LIN {X 0,Y 488.71,Z 151.612,A -85,B 0,C 180,E1 -6434.802,E2 -6434.802} C_VEL
LIN {X 0,Y 488.689,Z 151.612,A -85,B 0,C 180,E1 -6437.475,E2 -6437.475} C_VEL
LIN {X 0,Y 488.731,Z 151.607,A -85,B 0,C 180,E1 -6439.677,E2 -6439.677} C_VEL
LIN {X 0,Y 488.68,Z 151.615,A -85,B 0,C 180,E1 -6442.842,E2 -6442.842} C_VEL
LIN {X 0,Y 488.726,Z 151.608,A -85,B 0,C 180,E1 -6445.887,E2 -6445.887} C_VEL
LIN {X 0,Y 488.691,Z 151.614,A -85,B 0,C 180,E1 -6448.821,E2 -6448.821} C_VEL
LIN {X 0,Y 488.743,Z 151.606,A -85,B 0,C 180,E1 -6451.672,E2 -6451.672} C_VEL
LIN {X 0,Y 488.747,Z 151.606,A -85,B 0,C 180,E1 -6454.445,E2 -6454.445} C_VEL
LIN {X 0,Y 488.723,Z 151.609,A -85,B 0,C 180,E1 -6457.154,E2 -6457.154} C_VEL
LIN {X 0,Y 488.725,Z 151.608,A -85,B 0,C 180,E1 -6459.811,E2 -6459.811} C_VEL
LIN {X 0,Y 488.715,Z 151.612,A -85,B 0,C 180,E1 -6462.423,E2 -6462.423} C_VEL
LIN {X 0,Y 488.762,Z 151.603,A -85,B 0,C 180,E1 -6465,E2 -6465} C_VEL
LIN {X 0,Y 488.807,Z 151.601,A -85,B 0,C 180,E1 -6468.388,E2 -6468.388} C_VEL
LIN {X 0,Y 488.787,Z 151.6,A -85,B 0,C 180,E1 -6471.734,E2 -6471.734} C_VEL
LIN {X 0,Y 488.856,Z 151.594,A -85,B 0,C 180,E1 -6474.225,E2 -6474.225} C_VEL
LIN {X 0,Y 488.963,Z 151.578,A -85,B 0,C 180,E1 -6477.529,E2 -6477.529} C_VEL
LIN {X 0,Y 488.936,Z 151.581,A -85,B 0,C 180,E1 -6480.824,E2 -6480.824} C_VEL
LIN {X 0,Y 488.963,Z 151.579,A -85,B 0,C 180,E1 -6482.472,E2 -6482.472} C_VEL
LIN {X 0,Y 488.844,Z 151.594,A -85,B 0,C 180,E1 -6485.776,E2 -6485.776} C_VEL
LIN {X 0,Y 488.787,Z 151.601,A -85,B 0,C 180,E1 -6488.267,E2 -6488.267} C_VEL
LIN {X 0,Y 488.808,Z 151.6,A -85,B 0,C 180,E1 -6491.613,E2 -6491.613} C_VEL
LIN {X 0,Y 488.764,Z 151.604,A -85,B 0,C 180,E1 -6495.001,E2 -6495.001} C_VEL
LIN {X 0,Y 488.758,Z 151.605,A -85,B 0,C 180,E1 -6498.442,E2 -6498.442} C_VEL
LIN {X 0,Y 488.709,Z 151.611,A -85,B 0,C 180,E1 -6501.071,E2 -6501.071} C_VEL
LIN {X 0,Y 488.691,Z 151.613,A -85,B 0,C 180,E1 -6503.746,E2 -6503.746} C_VEL
LIN {X 0,Y 488.794,Z 151.6,A -85,B 0,C 180,E1 -6506.944,E2 -6506.944} C_VEL
LIN {X 0,Y 488.712,Z 151.61,A -85,B 0,C 180,E1 -6510.363,E2 -6510.363} C_VEL
LIN {X 0,Y 488.731,Z 151.608,A -85,B 0,C 180,E1 -6513.483,E2 -6513.483} C_VEL
LIN {X 0,Y 488.684,Z 151.612,A -85,B 0,C 180,E1 -6516.355,E2 -6516.355} C_VEL
LIN {X 0,Y 488.703,Z 151.613,A -85,B 0,C 180,E1 -6519.255,E2 -6519.255} C_VEL
LIN {X 0,Y 488.709,Z 151.611,A -85,B 0,C 180,E1 -6521.6,E2 -6521.6} C_VEL
LIN {X 0,Y 488.715,Z 151.607,A -85,B 0,C 180,E1 -6524.802,E2 -6524.802} C_VEL
LIN {X 0,Y 488.694,Z 151.611,A -85,B 0,C 180,E1 -6527.475,E2 -6527.475} C_VEL
LIN {X 0,Y 488.743,Z 151.622,A -85,B 0,C 180,E1 -6529.947,E2 -6529.947} C_VEL
LIN {X 0,Y 490.019,Z 158.689,A -85,B 0,C 180,E1 -6532.96,E2 -6532.96} C_VEL
LIN {X 0,Y 490.33,Z 163.252,A -85,B 0,C 180,E1 -6534.785,E2 -6534.785} C_VEL
LIN {X 0,Y 489.953,Z 171.835,A -85,B 0,C 180,E1 -6537.945,E2 -6537.945} C_VEL
LIN {X 0,Y 489.656,Z 178.453,A -85,B 0,C 180,E1 -6540.319,E2 -6540.319} C_VEL
LIN {X 0,Y 489.409,Z 185.796,A -85,B 0,C 180,E1 -6542.916,E2 -6542.916} C_VEL
LIN {X 0,Y 489.091,Z 194.423,A -85,B 0,C 180,E1 -6545.825,E2 -6545.825} C_VEL
LIN {X 0,Y 488.848,Z 204.699,A -85,B 0,C 180,E1 -6549.145,E2 -6549.145} C_VEL
LIN {X 0,Y 488.622,Z 213.613,A -85,B 0,C 180,E1 -6552.045,E2 -6552.045} C_VEL
LIN {X 0,Y 488.374,Z 223.582,A -85,B 0,C 180,E1 -6555.271,E2 -6555.271} C_VEL
LIN {X 0,Y 490.635,Z 237.098,A -85,B 0,C 180,E1 -6555.668,E2 -6555.668} C_VEL
LIN {X 0,Y 490.746,Z 245.176,A -85,B 0,C 180,E1 -6555.962,E2 -6555.962} C_VEL
LIN {X 0,Y 490.333,Z 257.492,A -85,B 0,C 180,E1 -6556.531,E2 -6556.531} C_VEL
LIN {X 0,Y 489.942,Z 269.529,A -85,B 0,C 180,E1 -6557.274,E2 -6557.274} C_VEL
LIN {X 0,Y 489.518,Z 281.094,A -85,B 0,C 180,E1 -6558.195,E2 -6558.195} C_VEL
LIN {X 0,Y 489.073,Z 291.54,A -85,B 0,C 180,E1 -6559.233,E2 -6559.233} C_VEL
LIN {X 0,Y 488.765,Z 299.992,A -85,B 0,C 180,E1 -6560.273,E2 -6560.273} C_VEL
LIN {X 0,Y 488.454,Z 308.236,A -85,B 0,C 180,E1 -6561.519,E2 -6561.519} C_VEL
LIN {X 0,Y 488.187,Z 314.876,A -85,B 0,C 180,E1 -6562.764,E2 -6562.764} C_VEL
LIN {X 0,Y 488.104,Z 320.95,A -85,B 0,C 180,E1 -6564.215,E2 -6564.215} C_VEL
LIN {X 0,Y 487.938,Z 324.895,A -85,B 0,C 180,E1 -6565.456,E2 -6565.456} C_VEL
LIN {X 0,Y 487.967,Z 327.807,A -85,B 0,C 180,E1 -6566.697,E2 -6566.697} C_VEL
LIN {X 0,Y 487.889,Z 330.183,A -85,B 0,C 180,E1 -6568.349,E2 -6568.349} C_VEL
LIN {X 0,Y 487.819,Z 331,A -85,B 0,C 180,E1 -6570,E2 -6570} C_VEL
LIN {X 0,Y 487.889,Z 330.184,A -85,B 0,C 180,E1 -6571.651,E2 -6571.651} C_VEL
LIN {X 0,Y 487.967,Z 327.81,A -85,B 0,C 180,E1 -6573.303,E2 -6573.303} C_VEL
LIN {X 0,Y 487.938,Z 324.895,A -85,B 0,C 180,E1 -6574.544,E2 -6574.544} C_VEL
LIN {X 0,Y 488.105,Z 320.948,A -85,B 0,C 180,E1 -6575.785,E2 -6575.785} C_VEL
LIN {X 0,Y 488.191,Z 314.875,A -85,B 0,C 180,E1 -6577.237,E2 -6577.237} C_VEL
LIN {X 0,Y 488.455,Z 308.235,A -85,B 0,C 180,E1 -6578.481,E2 -6578.481} C_VEL
LIN {X 0,Y 488.765,Z 299.99,A -85,B 0,C 180,E1 -6579.727,E2 -6579.727} C_VEL
LIN {X 0,Y 489.076,Z 291.538,A -85,B 0,C 180,E1 -6580.767,E2 -6580.767} C_VEL
LIN {X 0,Y 489.551,Z 281.09,A -85,B 0,C 180,E1 -6581.805,E2 -6581.805} C_VEL
LIN {X 0,Y 489.894,Z 269.887,A -85,B 0,C 180,E1 -6582.701,E2 -6582.701} C_VEL
LIN {X 0,Y 490.255,Z 259.402,A -85,B 0,C 180,E1 -6583.365,E2 -6583.365} C_VEL
LIN {X 0,Y 490.682,Z 247.759,A -85,B 0,C 180,E1 -6583.934,E2 -6583.934} C_VEL
LIN {X 0,Y 490.753,Z 237.916,A -85,B 0,C 180,E1 -6584.302,E2 -6584.302} C_VEL
LIN {X 0,Y 488.663,Z 225.221,A -85,B 0,C 180,E1 -6584.691,E2 -6584.691} C_VEL
LIN {X 0,Y 488.383,Z 223.53,A -85,B 0,C 180,E1 -6584.746,E2 -6584.746} C_VEL
LIN {X 0,Y 488.623,Z 213.612,A -85,B 0,C 180,E1 -6587.956,E2 -6587.956} C_VEL
LIN {X 0,Y 488.86,Z 204.014,A -85,B 0,C 180,E1 -6591.064,E2 -6591.064} C_VEL
LIN {X 0,Y 489.086,Z 194.276,A -85,B 0,C 180,E1 -6594.176,E2 -6594.176} C_VEL
LIN {X 0,Y 489.341,Z 185.619,A -85,B 0,C 180,E1 -6597.069,E2 -6597.069} C_VEL
LIN {X 0,Y 489.579,Z 178.064,A -85,B 0,C 180,E1 -6599.687,E2 -6599.687} C_VEL
LIN {X 0,Y 489.922,Z 170.008,A -85,B 0,C 180,E1 -6602.555,E2 -6602.555} C_VEL
LIN {X 0,Y 490.312,Z 162.957,A -85,B 0,C 180,E1 -6605.212,E2 -6605.212} C_VEL
LIN {X 0,Y 490.135,Z 159.545,A -85,B 0,C 180,E1 -6606.584,E2 -6606.584} C_VEL
LIN {X 0,Y 489.049,Z 153.497,A -85,B 0,C 180,E1 -6609.221,E2 -6609.221} C_VEL
LIN {X 0,Y 488.729,Z 151.611,A -85,B 0,C 180,E1 -6610.189,E2 -6610.189} C_VEL
LIN {X 0,Y 488.714,Z 151.609,A -85,B 0,C 180,E1 -6612.826,E2 -6612.826} C_VEL
LIN {X 0,Y 488.704,Z 151.613,A -85,B 0,C 180,E1 -6615.976,E2 -6615.976} C_VEL
LIN {X 0,Y 488.712,Z 151.614,A -85,B 0,C 180,E1 -6618.584,E2 -6618.584} C_VEL
LIN {X 0,Y 488.709,Z 151.613,A -85,B 0,C 180,E1 -6620.947,E2 -6620.947} C_VEL
LIN {X 0,Y 488.682,Z 151.615,A -85,B 0,C 180,E1 -6623.868,E2 -6623.868} C_VEL
LIN {X 0,Y 488.743,Z 151.607,A -85,B 0,C 180,E1 -6626.877,E2 -6626.877} C_VEL
LIN {X 0,Y 488.729,Z 151.609,A -85,B 0,C 180,E1 -6629.781,E2 -6629.781} C_VEL
LIN {X 0,Y 488.797,Z 151.6,A -85,B 0,C 180,E1 -6633.056,E2 -6633.056} C_VEL
LIN {X 0,Y 488.694,Z 151.614,A -85,B 0,C 180,E1 -6636.254,E2 -6636.254} C_VEL
LIN {X 0,Y 488.751,Z 151.606,A -85,B 0,C 180,E1 -6639.175,E2 -6639.175} C_VEL
LIN {X 0,Y 488.754,Z 151.605,A -85,B 0,C 180,E1 -6641.631,E2 -6641.631} C_VEL
LIN {X 0,Y 488.767,Z 151.603,A -85,B 0,C 180,E1 -6644.999,E2 -6644.999} C_VEL
LIN {X 0,Y 488.811,Z 151.6,A -85,B 0,C 180,E1 -6648.387,E2 -6648.387} C_VEL
LIN {X 0,Y 488.822,Z 151.598,A -85,B 0,C 180,E1 -6651.733,E2 -6651.733} C_VEL
LIN {X 0,Y 488.86,Z 151.592,A -85,B 0,C 180,E1 -6654.224,E2 -6654.224} C_VEL
LIN {X 0,Y 488.966,Z 151.58,A -85,B 0,C 180,E1 -6657.528,E2 -6657.528} C_VEL
LIN {X 0,Y 488.959,Z 151.581,A -85,B 0,C 180,E1 -6660.823,E2 -6660.823} C_VEL
LIN {X 0,Y 488.965,Z 151.58,A -85,B 0,C 180,E1 -6662.471,E2 -6662.471} C_VEL
LIN {X 0,Y 488.858,Z 151.595,A -85,B 0,C 180,E1 -6665.775,E2 -6665.775} C_VEL
LIN {X 0,Y 488.809,Z 151.6,A -85,B 0,C 180,E1 -6668.266,E2 -6668.266} C_VEL
LIN {X 0,Y 488.559,Z 151.634,A -85,B 0,C 180,E1 -6670.778,E2 -6670.778} C_VEL
LIN {X 0,Y 488.49,Z 151.748,A -85,B 0,C 180,E1 -6671.62,E2 -6671.62} C_VEL
LIN {X 0,Y 488.457,Z 155.39,A -85,B 0,C 180,E1 -6675.009,E2 -6675.009} C_VEL
LIN {X 0,Y 488.309,Z 159.042,A -85,B 0,C 180,E1 -6678.459,E2 -6678.459} C_VEL
LIN {X 0,Y 488.223,Z 161.933,A -85,B 0,C 180,E1 -6681.092,E2 -6681.092} C_VEL
LIN {X 0,Y 488.155,Z 164.836,A -85,B 0,C 180,E1 -6683.773,E2 -6683.773} C_VEL
LIN {X 0,Y 488.195,Z 168.106,A -85,B 0,C 180,E1 -6686.805,E2 -6686.805} C_VEL
LIN {X 0,Y 488.147,Z 170.848,A -85,B 0,C 180,E1 -6689.308,E2 -6689.308} C_VEL
LIN {X 0,Y 488.131,Z 172.135,A -85,B 0,C 180,E1 -6690.422,E2 -6690.422} C_VEL
LIN {X 0,Y 490.956,Z 184.643,A -85,B 0,C 180,E1 -6690.874,E2 -6690.874} C_VEL
LIN {X 0,Y 490.678,Z 197.29,A -85,B 0,C 180,E1 -6691.399,E2 -6691.399} C_VEL
LIN {X 0,Y 490.315,Z 208.569,A -85,B 0,C 180,E1 -6692.028,E2 -6692.028} C_VEL
LIN {X 0,Y 489.92,Z 219.575,A -85,B 0,C 180,E1 -6692.817,E2 -6692.817} C_VEL
LIN {X 0,Y 489.565,Z 230.593,A -85,B 0,C 180,E1 -6693.81,E2 -6693.81} C_VEL
LIN {X 0,Y 489.233,Z 239.42,A -85,B 0,C 180,E1 -6694.792,E2 -6694.792} C_VEL
LIN {X 0,Y 488.845,Z 247.344,A -85,B 0,C 180,E1 -6695.863,E2 -6695.863} C_VEL
LIN {X 0,Y 488.574,Z 255.122,A -85,B 0,C 180,E1 -6697.168,E2 -6697.168} C_VEL
LIN {X 0,Y 488.338,Z 261.885,A -85,B 0,C 180,E1 -6698.606,E2 -6698.606} C_VEL
LIN {X 0,Y 488.181,Z 266.165,A -85,B 0,C 180,E1 -6699.781,E2 -6699.781} C_VEL
LIN {X 0,Y 488.054,Z 269.408,A -85,B 0,C 180,E1 -6700.934,E2 -6700.934} C_VEL
LIN {X 0,Y 487.947,Z 272.607,A -85,B 0,C 180,E1 -6702.605,E2 -6702.605} C_VEL
LIN {X 0,Y 487.912,Z 273.948,A -85,B 0,C 180,E1 -6703.928,E2 -6703.928} C_VEL
LIN {X 0,Y 487.892,Z 274.307,A -85,B 0,C 180,E1 -6705.102,E2 -6705.102} C_VEL
LIN {X 0,Y 487.928,Z 273.85,A -85,B 0,C 180,E1 -6706.26,E2 -6706.26} C_VEL
LIN {X 0,Y 487.943,Z 272.646,A -85,B 0,C 180,E1 -6707.393,E2 -6707.393} C_VEL
LIN {X 0,Y 488.045,Z 269.503,A -85,B 0,C 180,E1 -6709.064,E2 -6709.064} C_VEL
LIN {X 0,Y 488.165,Z 266.271,A -85,B 0,C 180,E1 -6710.221,E2 -6710.221} C_VEL
LIN {X 0,Y 488.282,Z 262.041,A -85,B 0,C 180,E1 -6711.39,E2 -6711.39} C_VEL
LIN {X 0,Y 488.465,Z 256.703,A -85,B 0,C 180,E1 -6712.569,E2 -6712.569} C_VEL
LIN {X 0,Y 488.732,Z 249.328,A -85,B 0,C 180,E1 -6713.872,E2 -6713.872} C_VEL
LIN {X 0,Y 489.075,Z 241.461,A -85,B 0,C 180,E1 -6714.993,E2 -6714.993} C_VEL
LIN {X 0,Y 489.32,Z 235.534,A -85,B 0,C 180,E1 -6715.71,E2 -6715.71} C_VEL
LIN {X 0,Y 488.841,Z 231.28,A -85,B 0,C 180,E1 -6716.189,E2 -6716.189} C_VEL
LIN {X 0,Y 486.273,Z 224.218,A -85,B 0,C 180,E1 -6716.952,E2 -6716.952} C_VEL
LIN {X 0,Y 483.701,Z 216.705,A -85,B 0,C 180,E1 -6717.652,E2 -6717.652} C_VEL
LIN {X 0,Y 483.207,Z 211.749,A -85,B 0,C 180,E1 -6718.028,E2 -6718.028} C_VEL
LIN {X 0,Y 483.644,Z 199.873,A -85,B 0,C 180,E1 -6718.745,E2 -6718.745} C_VEL
LIN {X 0,Y 483.996,Z 188.065,A -85,B 0,C 180,E1 -6719.286,E2 -6719.286} C_VEL
LIN {X 0,Y 483.787,Z 184.103,A -85,B 0,C 180,E1 -6719.439,E2 -6719.439} C_VEL
LIN {X 0,Y 481.005,Z 171.659,A -85,B 0,C 180,E1 -6719.914,E2 -6719.914} C_VEL
LIN {X 0,Y 481.047,Z 168.051,A -85,B 0,C 180,E1 -6723.07,E2 -6723.07} C_VEL
LIN {X 0,Y 481.011,Z 164.908,A -85,B 0,C 180,E1 -6725.851,E2 -6725.851} C_VEL
LIN {X 0,Y 481.036,Z 161.858,A -85,B 0,C 180,E1 -6728.577,E2 -6728.577} C_VEL
LIN {X 0,Y 481.159,Z 158.393,A -85,B 0,C 180,E1 -6731.697,E2 -6731.697} C_VEL
LIN {X 0,Y 481.259,Z 155.027,A -85,B 0,C 180,E1 -6734.76,E2 -6734.76} C_VEL
LIN {X 0,Y 481.233,Z 153.146,A -85,B 0,C 180,E1 -6736.487,E2 -6736.487} C_VEL
LIN {X 0,Y 481.309,Z 152.535,A -85,B 0,C 180,E1 -6737.348,E2 -6737.348} C_VEL
LIN {X 0,Y 481.612,Z 152.497,A -85,B 0,C 180,E1 -6739.915,E2 -6739.915} C_VEL
LIN {X 0,Y 481.802,Z 152.472,A -85,B 0,C 180,E1 -6742.702,E2 -6742.702} C_VEL
LIN {X 0,Y 481.777,Z 152.474,A -85,B 0,C 180,E1 -6744.979,E2 -6744.979} C_VEL
LIN {X 0,Y 481.926,Z 152.456,A -85,B 0,C 180,E1 -6747.492,E2 -6747.492} C_VEL
LIN {X 0,Y 481.902,Z 152.458,A -85,B 0,C 180,E1 -6750.835,E2 -6750.835} C_VEL
LIN {X 0,Y 481.926,Z 152.455,A -85,B 0,C 180,E1 -6752.507,E2 -6752.507} C_VEL
LIN {X 0,Y 481.804,Z 152.472,A -85,B 0,C 180,E1 -6755.86,E2 -6755.86} C_VEL
LIN {X 0,Y 481.76,Z 152.477,A -85,B 0,C 180,E1 -6758.388,E2 -6758.388} C_VEL
LIN {X 0,Y 481.748,Z 152.479,A -85,B 0,C 180,E1 -6761.785,E2 -6761.785} C_VEL
LIN {X 0,Y 481.739,Z 152.478,A -85,B 0,C 180,E1 -6765.224,E2 -6765.224} C_VEL
LIN {X 0,Y 481.709,Z 152.48,A -85,B 0,C 180,E1 -6768.722,E2 -6768.722} C_VEL
LIN {X 0,Y 481.645,Z 152.491,A -85,B 0,C 180,E1 -6771.395,E2 -6771.395} C_VEL
LIN {X 0,Y 481.675,Z 152.487,A -85,B 0,C 180,E1 -6774.113,E2 -6774.113} C_VEL
LIN {X 0,Y 481.744,Z 152.478,A -85,B 0,C 180,E1 -6777.139,E2 -6777.139} C_VEL
LIN {X 0,Y 481.676,Z 152.487,A -85,B 0,C 180,E1 -6779.741,E2 -6779.741} C_VEL
LIN {X 0,Y 481.669,Z 152.488,A -85,B 0,C 180,E1 -6782.674,E2 -6782.674} C_VEL
LIN {X 0,Y 481.633,Z 152.492,A -85,B 0,C 180,E1 -6785.71,E2 -6785.71} C_VEL
LIN {X 0,Y 481.669,Z 152.489,A -85,B 0,C 180,E1 -6788.859,E2 -6788.859} C_VEL
LIN {X 0,Y 481.651,Z 152.49,A -85,B 0,C 180,E1 -6791.913,E2 -6791.913} C_VEL
LIN {X 0,Y 481.657,Z 152.488,A -85,B 0,C 180,E1 -6794.458,E2 -6794.458} C_VEL
LIN {X 0,Y 481.645,Z 152.49,A -85,B 0,C 180,E1 -6797.84,E2 -6797.84} C_VEL
LIN {X 0,Y 481.679,Z 152.488,A -85,B 0,C 180,E1 -6800.652,E2 -6800.652} C_VEL
LIN {X 0,Y 481.629,Z 152.492,A -85,B 0,C 180,E1 -6803.376,E2 -6803.376} C_VEL
LIN {X 0,Y 481.692,Z 152.484,A -85,B 0,C 180,E1 -6806.329,E2 -6806.329} C_VEL
LIN {X 0,Y 481.649,Z 152.488,A -85,B 0,C 180,E1 -6809.418,E2 -6809.418} C_VEL
LIN {X 0,Y 481.699,Z 152.483,A -85,B 0,C 180,E1 -6812.169,E2 -6812.169} C_VEL
LIN {X 0,Y 481.717,Z 152.484,A -85,B 0,C 180,E1 -6814.97,E2 -6814.97} C_VEL
LIN {X 0,Y 481.649,Z 152.49,A -85,B 0,C 180,E1 -6817.705,E2 -6817.705} C_VEL
LIN {X 0,Y 481.705,Z 152.484,A -85,B 0,C 180,E1 -6820.394,E2 -6820.394} C_VEL
LIN {X 0,Y 481.679,Z 152.486,A -85,B 0,C 180,E1 -6823.034,E2 -6823.034} C_VEL
LIN {X 0,Y 481.689,Z 152.483,A -85,B 0,C 180,E1 -6825.639,E2 -6825.639} C_VEL
LIN {X 0,Y 481.752,Z 152.478,A -85,B 0,C 180,E1 -6828.216,E2 -6828.216} C_VEL
LIN {X 0,Y 481.742,Z 152.477,A -85,B 0,C 180,E1 -6831.612,E2 -6831.612} C_VEL
LIN {X 0,Y 481.817,Z 152.47,A -85,B 0,C 180,E1 -6834.14,E2 -6834.14} C_VEL
LIN {X 0,Y 481.93,Z 152.454,A -85,B 0,C 180,E1 -6837.493,E2 -6837.493} C_VEL
LIN {X 0,Y 481.888,Z 152.459,A -85,B 0,C 180,E1 -6840.836,E2 -6840.836} C_VEL
LIN {X 0,Y 481.93,Z 152.455,A -85,B 0,C 180,E1 -6842.508,E2 -6842.508} C_VEL
LIN {X 0,Y 481.802,Z 152.471,A -85,B 0,C 180,E1 -6845.861,E2 -6845.861} C_VEL
LIN {X 0,Y 481.742,Z 152.478,A -85,B 0,C 180,E1 -6848.389,E2 -6848.389} C_VEL
LIN {X 0,Y 481.753,Z 152.478,A -85,B 0,C 180,E1 -6851.785,E2 -6851.785} C_VEL
LIN {X 0,Y 481.745,Z 152.48,A -85,B 0,C 180,E1 -6855.225,E2 -6855.225} C_VEL
LIN {X 0,Y 481.715,Z 152.482,A -85,B 0,C 180,E1 -6858.722,E2 -6858.722} C_VEL
LIN {X 0,Y 481.648,Z 152.491,A -85,B 0,C 180,E1 -6861.395,E2 -6861.395} C_VEL
LIN {X 0,Y 481.676,Z 152.486,A -85,B 0,C 180,E1 -6864.114,E2 -6864.114} C_VEL
LIN {X 0,Y 481.749,Z 152.479,A -85,B 0,C 180,E1 -6867.139,E2 -6867.139} C_VEL
LIN {X 0,Y 481.681,Z 152.486,A -85,B 0,C 180,E1 -6869.741,E2 -6869.741} C_VEL
LIN {X 0,Y 481.673,Z 152.486,A -85,B 0,C 180,E1 -6872.675,E2 -6872.675} C_VEL
LIN {X 0,Y 481.638,Z 152.491,A -85,B 0,C 180,E1 -6875.71,E2 -6875.71} C_VEL
LIN {X 0,Y 481.673,Z 152.487,A -85,B 0,C 180,E1 -6878.859,E2 -6878.859} C_VEL
LIN {X 0,Y 481.655,Z 152.488,A -85,B 0,C 180,E1 -6881.913,E2 -6881.913} C_VEL
LIN {X 0,Y 481.662,Z 152.485,A -85,B 0,C 180,E1 -6884.458,E2 -6884.458} C_VEL
LIN {X 0,Y 481.65,Z 152.489,A -85,B 0,C 180,E1 -6887.84,E2 -6887.84} C_VEL
LIN {X 0,Y 481.691,Z 152.571,A -85,B 0,C 180,E1 -6889.67,E2 -6889.67} C_VEL
LIN {X 0,Y 482.777,Z 158.616,A -85,B 0,C 180,E1 -6892.308,E2 -6892.308} C_VEL
LIN {X 0,Y 483.312,Z 162.509,A -85,B 0,C 180,E1 -6893.919,E2 -6893.919} C_VEL
LIN {X 0,Y 483.176,Z 167.84,A -85,B 0,C 180,E1 -6896.006,E2 -6896.006} C_VEL
LIN {X 0,Y 482.822,Z 176.447,A -85,B 0,C 180,E1 -6899.184,E2 -6899.184} C_VEL
LIN {X 0,Y 482.425,Z 186.22,A -85,B 0,C 180,E1 -6902.705,E2 -6902.705} C_VEL
LIN {X 0,Y 482.026,Z 195.527,A -85,B 0,C 180,E1 -6905.906,E2 -6905.906} C_VEL
LIN {X 0,Y 481.797,Z 204.962,A -85,B 0,C 180,E1 -6908.999,E2 -6908.999} C_VEL
LIN {X 0,Y 481.551,Z 214.717,A -85,B 0,C 180,E1 -6912.153,E2 -6912.153} C_VEL
LIN {X 0,Y 481.333,Z 223.582,A -85,B 0,C 180,E1 -6915.05,E2 -6915.05} C_VEL
LIN {X 0,Y 483.642,Z 237.098,A -85,B 0,C 180,E1 -6915.456,E2 -6915.456} C_VEL
LIN {X 0,Y 483.902,Z 242.504,A -85,B 0,C 180,E1 -6915.652,E2 -6915.652} C_VEL
LIN {X 0,Y 483.564,Z 254.512,A -85,B 0,C 180,E1 -6916.179,E2 -6916.179} C_VEL
LIN {X 0,Y 483.131,Z 266.185,A -85,B 0,C 180,E1 -6916.861,E2 -6916.861} C_VEL
LIN {X 0,Y 482.726,Z 277.486,A -85,B 0,C 180,E1 -6917.706,E2 -6917.706} C_VEL
LIN {X 0,Y 482.313,Z 287.647,A -85,B 0,C 180,E1 -6918.655,E2 -6918.655} C_VEL
LIN {X 0,Y 481.877,Z 296.786,A -85,B 0,C 180,E1 -6919.708,E2 -6919.708} C_VEL
LIN {X 0,Y 481.531,Z 305.688,A -85,B 0,C 180,E1 -6920.973,E2 -6920.973} C_VEL
LIN {X 0,Y 481.208,Z 312.849,A -85,B 0,C 180,E1 -6922.236,E2 -6922.236} C_VEL
LIN {X 0,Y 481.045,Z 318.374,A -85,B 0,C 180,E1 -6923.452,E2 -6923.452} C_VEL
LIN {X 0,Y 480.999,Z 322.373,A -85,B 0,C 180,E1 -6924.55,E2 -6924.55} C_VEL
LIN {X 0,Y 480.847,Z 325.958,A -85,B 0,C 180,E1 -6925.809,E2 -6925.809} C_VEL
LIN {X 0,Y 480.892,Z 327.807,A -85,B 0,C 180,E1 -6926.649,E2 -6926.649} C_VEL
LIN {X 0,Y 480.79,Z 330.182,A -85,B 0,C 180,E1 -6928.325,E2 -6928.325} C_VEL
LIN {X 0,Y 480.743,Z 331,A -85,B 0,C 180,E1 -6930,E2 -6930} C_VEL
LIN {X 0,Y 480.79,Z 330.184,A -85,B 0,C 180,E1 -6931.675,E2 -6931.675} C_VEL
LIN {X 0,Y 480.892,Z 327.81,A -85,B 0,C 180,E1 -6933.351,E2 -6933.351} C_VEL
LIN {X 0,Y 480.854,Z 324.895,A -85,B 0,C 180,E1 -6934.611,E2 -6934.611} C_VEL
LIN {X 0,Y 481.023,Z 320.948,A -85,B 0,C 180,E1 -6935.87,E2 -6935.87} C_VEL
LIN {X 0,Y 481.117,Z 314.875,A -85,B 0,C 180,E1 -6937.344,E2 -6937.344} C_VEL
LIN {X 0,Y 481.427,Z 308.234,A -85,B 0,C 180,E1 -6938.606,E2 -6938.606} C_VEL
LIN {X 0,Y 481.757,Z 299.991,A -85,B 0,C 180,E1 -6939.87,E2 -6939.87} C_VEL
LIN {X 0,Y 482.081,Z 291.538,A -85,B 0,C 180,E1 -6940.925,E2 -6940.925} C_VEL
LIN {X 0,Y 482.586,Z 281.089,A -85,B 0,C 180,E1 -6941.978,E2 -6941.978} C_VEL
LIN {X 0,Y 482.969,Z 269.875,A -85,B 0,C 180,E1 -6942.887,E2 -6942.887} C_VEL
LIN {X 0,Y 483.348,Z 259.401,A -85,B 0,C 180,E1 -6943.56,E2 -6943.56} C_VEL
LIN {X 0,Y 483.801,Z 247.759,A -85,B 0,C 180,E1 -6944.136,E2 -6944.136} C_VEL
LIN {X 0,Y 483.801,Z 238.298,A -85,B 0,C 180,E1 -6944.499,E2 -6944.499} C_VEL
LIN {X 0,Y 481.632,Z 225.324,A -85,B 0,C 180,E1 -6944.908,E2 -6944.908} C_VEL
LIN {X 0,Y 481.325,Z 223.53,A -85,B 0,C 180,E1 -6944.967,E2 -6944.967} C_VEL
LIN {X 0,Y 481.552,Z 214.708,A -85,B 0,C 180,E1 -6947.848,E2 -6947.848} C_VEL
LIN {X 0,Y 481.797,Z 204.857,A -85,B 0,C 180,E1 -6951.001,E2 -6951.001} C_VEL
LIN {X 0,Y 482.022,Z 195.31,A -85,B 0,C 180,E1 -6954.095,E2 -6954.095} C_VEL
LIN {X 0,Y 482.336,Z 185.992,A -85,B 0,C 180,E1 -6957.274,E2 -6957.274} C_VEL
LIN {X 0,Y 482.626,Z 177.805,A -85,B 0,C 180,E1 -6960.158,E2 -6960.158} C_VEL
LIN {X 0,Y 483.012,Z 169.886,A -85,B 0,C 180,E1 -6963.069,E2 -6963.069} C_VEL
LIN {X 0,Y 483.33,Z 163.415,A -85,B 0,C 180,E1 -6965.566,E2 -6965.566} C_VEL
LIN {X 0,Y 483.091,Z 160.328,A -85,B 0,C 180,E1 -6966.856,E2 -6966.856} C_VEL
LIN {X 0,Y 481.884,Z 153.509,A -85,B 0,C 180,E1 -6969.92,E2 -6969.92} C_VEL
LIN {X 0,Y 481.689,Z 152.488,A -85,B 0,C 180,E1 -6970.462,E2 -6970.462} C_VEL
LIN {X 0,Y 481.644,Z 152.489,A -85,B 0,C 180,E1 -6973.3,E2 -6973.3} C_VEL
LIN {X 0,Y 481.663,Z 152.49,A -85,B 0,C 180,E1 -6975.641,E2 -6975.641} C_VEL
LIN {X 0,Y 481.661,Z 152.492,A -85,B 0,C 180,E1 -6978.958,E2 -6978.958} C_VEL
LIN {X 0,Y 481.659,Z 152.491,A -85,B 0,C 180,E1 -6981.993,E2 -6981.993} C_VEL
LIN {X 0,Y 481.693,Z 152.486,A -85,B 0,C 180,E1 -6985.318,E2 -6985.318} C_VEL
LIN {X 0,Y 481.651,Z 152.492,A -85,B 0,C 180,E1 -6988.312,E2 -6988.312} C_VEL
LIN {X 0,Y 481.705,Z 152.483,A -85,B 0,C 180,E1 -6991.218,E2 -6991.218} C_VEL
LIN {X 0,Y 481.706,Z 152.484,A -85,B 0,C 180,E1 -6994.043,E2 -6994.043} C_VEL
LIN {X 0,Y 481.679,Z 152.487,A -85,B 0,C 180,E1 -6996.812,E2 -6996.812} C_VEL
LIN {X 0,Y 481.7,Z 152.484,A -85,B 0,C 180,E1 -6999.503,E2 -6999.503} C_VEL
LIN {X 0,Y 481.696,Z 152.483,A -85,B 0,C 180,E1 -7002.158,E2 -7002.158} C_VEL
LIN {X 0,Y 481.748,Z 152.478,A -85,B 0,C 180,E1 -7004.776,E2 -7004.776} C_VEL
LIN {X 0,Y 481.756,Z 152.478,A -85,B 0,C 180,E1 -7008.215,E2 -7008.215} C_VEL
LIN {X 0,Y 481.768,Z 152.477,A -85,B 0,C 180,E1 -7011.611,E2 -7011.611} C_VEL
LIN {X 0,Y 481.821,Z 152.469,A -85,B 0,C 180,E1 -7014.139,E2 -7014.139} C_VEL
LIN {X 0,Y 481.933,Z 152.456,A -85,B 0,C 180,E1 -7017.492,E2 -7017.492} C_VEL
LIN {X 0,Y 481.91,Z 152.458,A -85,B 0,C 180,E1 -7020.835,E2 -7020.835} C_VEL
LIN {X 0,Y 481.932,Z 152.456,A -85,B 0,C 180,E1 -7022.507,E2 -7022.507} C_VEL
LIN {X 0,Y 481.82,Z 152.472,A -85,B 0,C 180,E1 -7025.86,E2 -7025.86} C_VEL
LIN {X 0,Y 481.752,Z 152.48,A -85,B 0,C 180,E1 -7028.388,E2 -7028.388} C_VEL
LIN {X 0,Y 481.511,Z 152.512,A -85,B 0,C 180,E1 -7030.937,E2 -7030.937} C_VEL
LIN {X 0,Y 481.456,Z 153.051,A -85,B 0,C 180,E1 -7032.032,E2 -7032.032} C_VEL
LIN {X 0,Y 481.381,Z 156.725,A -85,B 0,C 180,E1 -7035.51,E2 -7035.51} C_VEL
LIN {X 0,Y 481.246,Z 160.17,A -85,B 0,C 180,E1 -7038.74,E2 -7038.74} C_VEL
LIN {X 0,Y 481.157,Z 163.021,A -85,B 0,C 180,E1 -7041.417,E2 -7041.417} C_VEL
LIN {X 0,Y 481.108,Z 165.967,A -85,B 0,C 180,E1 -7044.143,E2 -7044.143} C_VEL
LIN {X 0,Y 481.125,Z 169.043,A -85,B 0,C 180,E1 -7046.993,E2 -7046.993} C_VEL
LIN {X 0,Y 481.083,Z 172.545,A -85,B 0,C 180,E1 -7050.198,E2 -7050.198} C_VEL
LIN {X 0,Y 484.078,Z 185.544,A -85,B 0,C 180,E1 -7050.685,E2 -7050.685} C_VEL
LIN {X 0,Y 483.795,Z 197.865,A -85,B 0,C 180,E1 -7051.209,E2 -7051.209} C_VEL
LIN {X 0,Y 483.452,Z 208.374,A -85,B 0,C 180,E1 -7051.8,E2 -7051.8} C_VEL
LIN {X 0,Y 483.038,Z 219.144,A -85,B 0,C 180,E1 -7052.57,E2 -7052.57} C_VEL
LIN {X 0,Y 482.636,Z 230.505,A -85,B 0,C 180,E1 -7053.596,E2 -7053.596} C_VEL
LIN {X 0,Y 482.268,Z 239.774,A -85,B 0,C 180,E1 -7054.634,E2 -7054.634} C_VEL
LIN {X 0,Y 481.859,Z 247.523,A -85,B 0,C 180,E1 -7055.69,E2 -7055.69} C_VEL
LIN {X 0,Y 481.563,Z 255.349,A -85,B 0,C 180,E1 -7057.013,E2 -7057.013} C_VEL
LIN {X 0,Y 481.325,Z 261.835,A -85,B 0,C 180,E1 -7058.397,E2 -7058.397} C_VEL
LIN {X 0,Y 481.122,Z 266.265,A -85,B 0,C 180,E1 -7059.604,E2 -7059.604} C_VEL
LIN {X 0,Y 480.978,Z 270.412,A -85,B 0,C 180,E1 -7061.112,E2 -7061.112} C_VEL
LIN {X 0,Y 480.872,Z 272.569,A -85,B 0,C 180,E1 -7062.244,E2 -7062.244} C_VEL
LIN {X 0,Y 480.846,Z 273.976,A -85,B 0,C 180,E1 -7063.388,E2 -7063.388} C_VEL
LIN {X 0,Y 480.803,Z 274.666,A -85,B 0,C 180,E1 -7064.557,E2 -7064.557} C_VEL
LIN {X 0,Y 480.809,Z 274.59,A -85,B 0,C 180,E1 -7065.744,E2 -7065.744} C_VEL
LIN {X 0,Y 480.873,Z 273.669,A -85,B 0,C 180,E1 -7066.949,E2 -7066.949} C_VEL
LIN {X 0,Y 480.896,Z 271.865,A -85,B 0,C 180,E1 -7068.187,E2 -7068.187} C_VEL
LIN {X 0,Y 481.004,Z 269.102,A -85,B 0,C 180,E1 -7069.444,E2 -7069.444} C_VEL
LIN {X 0,Y 481.152,Z 265.238,A -85,B 0,C 180,E1 -7070.727,E2 -7070.727} C_VEL
LIN {X 0,Y 481.384,Z 259.475,A -85,B 0,C 180,E1 -7072.18,E2 -7072.18} C_VEL
LIN {X 0,Y 481.643,Z 252.032,A -85,B 0,C 180,E1 -7073.614,E2 -7073.614} C_VEL
LIN {X 0,Y 481.988,Z 243.638,A -85,B 0,C 180,E1 -7074.9,E2 -7074.9} C_VEL
LIN {X 0,Y 482.386,Z 234.709,A -85,B 0,C 180,E1 -7076,E2 -7076} C_VEL
LIN {X 0,Y 482.775,Z 224.312,A -85,B 0,C 180,E1 -7077.037,E2 -7077.037} C_VEL
LIN {X 0,Y 483.162,Z 213.156,A -85,B 0,C 180,E1 -7077.932,E2 -7077.932} C_VEL
LIN {X 0,Y 483.207,Z 211.749,A -85,B 0,C 180,E1 -7078.028,E2 -7078.028} C_VEL
LIN {X 0,Y 482.64,Z 204.929,A -85,B 0,C 180,E1 -7078.488,E2 -7078.488} C_VEL
LIN {X 0,Y 480.926,Z 198.148,A -85,B 0,C 180,E1 -7078.924,E2 -7078.924} C_VEL
LIN {X 0,Y 478.679,Z 191.263,A -85,B 0,C 180,E1 -7079.321,E2 -7079.321} C_VEL
LIN {X 0,Y 476.664,Z 184.126,A -85,B 0,C 180,E1 -7079.667,E2 -7079.667} C_VEL
LIN {X 0,Y 473.917,Z 172.054,A -85,B 0,C 180,E1 -7080.12,E2 -7080.12} C_VEL
LIN {X 0,Y 473.971,Z 168.106,A -85,B 0,C 180,E1 -7083.587,E2 -7083.587} C_VEL
LIN {X 0,Y 473.967,Z 164.475,A -85,B 0,C 180,E1 -7086.828,E2 -7086.828} C_VEL
LIN {X 0,Y 474.007,Z 160.896,A -85,B 0,C 180,E1 -7090.061,E2 -7090.061} C_VEL
LIN {X 0,Y 474.1,Z 157.945,A -85,B 0,C 180,E1 -7092.754,E2 -7092.754} C_VEL
LIN {X 0,Y 474.179,Z 155.051,A -85,B 0,C 180,E1 -7095.406,E2 -7095.406} C_VEL
LIN {X 0,Y 474.24,Z 153.415,A -85,B 0,C 180,E1 -7097.156,E2 -7097.156} C_VEL
LIN {X 0,Y 474.546,Z 153.376,A -85,B 0,C 180,E1 -7099.763,E2 -7099.763} C_VEL
LIN {X 0,Y 474.752,Z 153.35,A -85,B 0,C 180,E1 -7102.669,E2 -7102.669} C_VEL
LIN {X 0,Y 474.747,Z 153.35,A -85,B 0,C 180,E1 -7104.904,E2 -7104.904} C_VEL
LIN {X 0,Y 474.892,Z 153.331,A -85,B 0,C 180,E1 -7107.455,E2 -7107.455} C_VEL
LIN {X 0,Y 474.909,Z 153.332,A -85,B 0,C 180,E1 -7110,E2 -7110} C_VEL
LIN {X 0,Y 474.892,Z 153.331,A -85,B 0,C 180,E1 -7112.544,E2 -7112.544} C_VEL
LIN {X 0,Y 474.767,Z 153.35,A -85,B 0,C 180,E1 -7115.948,E2 -7115.948} C_VEL
LIN {X 0,Y 474.725,Z 153.352,A -85,B 0,C 180,E1 -7118.513,E2 -7118.513} C_VEL
LIN {X 0,Y 474.701,Z 153.358,A -85,B 0,C 180,E1 -7121.962,E2 -7121.962} C_VEL
LIN {X 0,Y 474.697,Z 153.357,A -85,B 0,C 180,E1 -7125.456,E2 -7125.456} C_VEL
LIN {X 0,Y 474.662,Z 153.359,A -85,B 0,C 180,E1 -7129.01,E2 -7129.01} C_VEL
LIN {X 0,Y 474.587,Z 153.371,A -85,B 0,C 180,E1 -7131.729,E2 -7131.729} C_VEL
LIN {X 0,Y 474.656,Z 153.36,A -85,B 0,C 180,E1 -7134.493,E2 -7134.493} C_VEL
LIN {X 0,Y 474.696,Z 153.357,A -85,B 0,C 180,E1 -7137.339,E2 -7137.339} C_VEL
LIN {X 0,Y 474.601,Z 153.367,A -85,B 0,C 180,E1 -7140.81,E2 -7140.81} C_VEL
LIN {X 0,Y 474.634,Z 153.363,A -85,B 0,C 180,E1 -7143.984,E2 -7143.984} C_VEL
LIN {X 0,Y 474.569,Z 153.372,A -85,B 0,C 180,E1 -7146.9,E2 -7146.9} C_VEL
LIN {X 0,Y 474.625,Z 153.366,A -85,B 0,C 180,E1 -7149.648,E2 -7149.648} C_VEL
LIN {X 0,Y 474.613,Z 153.367,A -85,B 0,C 180,E1 -7152.934,E2 -7152.934} C_VEL
LIN {X 0,Y 474.607,Z 153.367,A -85,B 0,C 180,E1 -7155.896,E2 -7155.896} C_VEL
LIN {X 0,Y 474.625,Z 153.366,A -85,B 0,C 180,E1 -7159.041,E2 -7159.041} C_VEL
LIN {X 0,Y 474.609,Z 153.367,A -85,B 0,C 180,E1 -7161.704,E2 -7161.704} C_VEL
LIN {X 0,Y 474.625,Z 153.366,A -85,B 0,C 180,E1 -7164.726,E2 -7164.726} C_VEL
LIN {X 0,Y 474.633,Z 153.363,A -85,B 0,C 180,E1 -7167.788,E2 -7167.788} C_VEL
LIN {X 0,Y 474.622,Z 153.366,A -85,B 0,C 180,E1 -7170.885,E2 -7170.885} C_VEL
LIN {X 0,Y 474.66,Z 153.36,A -85,B 0,C 180,E1 -7173.629,E2 -7173.629} C_VEL
LIN {X 0,Y 474.635,Z 153.365,A -85,B 0,C 180,E1 -7176.642,E2 -7176.642} C_VEL
LIN {X 0,Y 474.655,Z 153.363,A -85,B 0,C 180,E1 -7180.09,E2 -7180.09} C_VEL
LIN {X 0,Y 474.639,Z 153.363,A -85,B 0,C 180,E1 -7182.775,E2 -7182.775} C_VEL
LIN {X 0,Y 474.647,Z 153.36,A -85,B 0,C 180,E1 -7185.421,E2 -7185.421} C_VEL
LIN {X 0,Y 474.705,Z 153.355,A -85,B 0,C 180,E1 -7188.038,E2 -7188.038} C_VEL
LIN {X 0,Y 474.714,Z 153.353,A -85,B 0,C 180,E1 -7191.487,E2 -7191.487} C_VEL
LIN {X 0,Y 474.78,Z 153.346,A -85,B 0,C 180,E1 -7194.053,E2 -7194.053} C_VEL
LIN {X 0,Y 474.896,Z 153.331,A -85,B 0,C 180,E1 -7197.456,E2 -7197.456} C_VEL
LIN {X 0,Y 474.914,Z 153.329,A -85,B 0,C 180,E1 -7200,E2 -7200} C_VEL
LIN {X 0,Y 474.896,Z 153.332,A -85,B 0,C 180,E1 -7202.545,E2 -7202.545} C_VEL
LIN {X 0,Y 474.763,Z 153.348,A -85,B 0,C 180,E1 -7205.948,E2 -7205.948} C_VEL
LIN {X 0,Y 474.713,Z 153.354,A -85,B 0,C 180,E1 -7208.514,E2 -7208.514} C_VEL
LIN {X 0,Y 474.707,Z 153.355,A -85,B 0,C 180,E1 -7211.963,E2 -7211.963} C_VEL
LIN {X 0,Y 474.702,Z 153.356,A -85,B 0,C 180,E1 -7215.456,E2 -7215.456} C_VEL
LIN {X 0,Y 474.667,Z 153.36,A -85,B 0,C 180,E1 -7219.011,E2 -7219.011} C_VEL
LIN {X 0,Y 474.591,Z 153.37,A -85,B 0,C 180,E1 -7221.729,E2 -7221.729} C_VEL
LIN {X 0,Y 474.659,Z 153.36,A -85,B 0,C 180,E1 -7224.493,E2 -7224.493} C_VEL
LIN {X 0,Y 474.684,Z 153.359,A -85,B 0,C 180,E1 -7227.335,E2 -7227.335} C_VEL
LIN {X 0,Y 474.607,Z 153.368,A -85,B 0,C 180,E1 -7230.81,E2 -7230.81} C_VEL
LIN {X 0,Y 474.627,Z 153.367,A -85,B 0,C 180,E1 -7233.222,E2 -7233.222} C_VEL
LIN {X 0,Y 474.591,Z 153.368,A -85,B 0,C 180,E1 -7236.324,E2 -7236.324} C_VEL
LIN {X 0,Y 474.62,Z 153.365,A -85,B 0,C 180,E1 -7239.646,E2 -7239.646} C_VEL
LIN {X 0,Y 474.617,Z 153.364,A -85,B 0,C 180,E1 -7242.934,E2 -7242.934} C_VEL
LIN {X 0,Y 474.611,Z 153.363,A -85,B 0,C 180,E1 -7245.895,E2 -7245.895} C_VEL
LIN {X 0,Y 474.629,Z 153.365,A -85,B 0,C 180,E1 -7249.192,E2 -7249.192} C_VEL
LIN {X 0,Y 474.624,Z 153.402,A -85,B 0,C 180,E1 -7249.343,E2 -7249.343} C_VEL
LIN {X 0,Y 475.788,Z 159.819,A -85,B 0,C 180,E1 -7252.193,E2 -7252.193} C_VEL
LIN {X 0,Y 476.33,Z 163.704,A -85,B 0,C 180,E1 -7253.83,E2 -7253.83} C_VEL
LIN {X 0,Y 476.2,Z 168.886,A -85,B 0,C 180,E1 -7255.887,E2 -7255.887} C_VEL
LIN {X 0,Y 475.84,Z 176.962,A -85,B 0,C 180,E1 -7258.942,E2 -7258.942} C_VEL
LIN {X 0,Y 475.416,Z 186.67,A -85,B 0,C 180,E1 -7262.496,E2 -7262.496} C_VEL
LIN {X 0,Y 475.027,Z 195.252,A -85,B 0,C 180,E1 -7265.527,E2 -7265.527} C_VEL
LIN {X 0,Y 474.752,Z 205.221,A -85,B 0,C 180,E1 -7268.848,E2 -7268.848} C_VEL
LIN {X 0,Y 474.49,Z 214.451,A -85,B 0,C 180,E1 -7271.878,E2 -7271.878} C_VEL
LIN {X 0,Y 474.292,Z 223.632,A -85,B 0,C 180,E1 -7274.827,E2 -7274.827} C_VEL
LIN {X 0,Y 476.609,Z 237.098,A -85,B 0,C 180,E1 -7275.237,E2 -7275.237} C_VEL
LIN {X 0,Y 477.045,Z 242.505,A -85,B 0,C 180,E1 -7275.441,E2 -7275.441} C_VEL
LIN {X 0,Y 476.63,Z 255.504,A -85,B 0,C 180,E1 -7276.028,E2 -7276.028} C_VEL
LIN {X 0,Y 476.186,Z 266.678,A -85,B 0,C 180,E1 -7276.7,E2 -7276.7} C_VEL
LIN {X 0,Y 475.781,Z 277.485,A -85,B 0,C 180,E1 -7277.524,E2 -7277.524} C_VEL
LIN {X 0,Y 475.356,Z 287.647,A -85,B 0,C 180,E1 -7278.487,E2 -7278.487} C_VEL
LIN {X 0,Y 474.878,Z 296.786,A -85,B 0,C 180,E1 -7279.555,E2 -7279.555} C_VEL
LIN {X 0,Y 474.483,Z 305.688,A -85,B 0,C 180,E1 -7280.838,E2 -7280.838} C_VEL
LIN {X 0,Y 474.153,Z 312.849,A -85,B 0,C 180,E1 -7282.12,E2 -7282.12} C_VEL
LIN {X 0,Y 473.973,Z 318.739,A -85,B 0,C 180,E1 -7283.449,E2 -7283.449} C_VEL
LIN {X 0,Y 473.846,Z 323.677,A -85,B 0,C 180,E1 -7284.895,E2 -7284.895} C_VEL
LIN {X 0,Y 473.752,Z 325.958,A -85,B 0,C 180,E1 -7285.746,E2 -7285.746} C_VEL
LIN {X 0,Y 473.8,Z 327.807,A -85,B 0,C 180,E1 -7286.599,E2 -7286.599} C_VEL
LIN {X 0,Y 473.695,Z 330.182,A -85,B 0,C 180,E1 -7288.3,E2 -7288.3} C_VEL
LIN {X 0,Y 473.688,Z 330.786,A -85,B 0,C 180,E1 -7289.15,E2 -7289.15} C_VEL
LIN {X 0,Y 473.669,Z 331,A -85,B 0,C 180,E1 -7290,E2 -7290} C_VEL
LIN {X 0,Y 473.688,Z 330.786,A -85,B 0,C 180,E1 -7290.85,E2 -7290.85} C_VEL
LIN {X 0,Y 473.724,Z 329.196,A -85,B 0,C 180,E1 -7292.551,E2 -7292.551} C_VEL
LIN {X 0,Y 473.8,Z 327.81,A -85,B 0,C 180,E1 -7293.402,E2 -7293.402} C_VEL
LIN {X 0,Y 473.776,Z 324.895,A -85,B 0,C 180,E1 -7294.68,E2 -7294.68} C_VEL
LIN {X 0,Y 473.943,Z 320.947,A -85,B 0,C 180,E1 -7295.958,E2 -7295.958} C_VEL
LIN {X 0,Y 474.05,Z 314.875,A -85,B 0,C 180,E1 -7297.454,E2 -7297.454} C_VEL
LIN {X 0,Y 474.378,Z 308.234,A -85,B 0,C 180,E1 -7298.735,E2 -7298.735} C_VEL
LIN {X 0,Y 474.752,Z 299.991,A -85,B 0,C 180,E1 -7300.017,E2 -7300.017} C_VEL
LIN {X 0,Y 475.098,Z 291.538,A -85,B 0,C 180,E1 -7301.088,E2 -7301.088} C_VEL
LIN {X 0,Y 475.631,Z 281.11,A -85,B 0,C 180,E1 -7302.153,E2 -7302.153} C_VEL
LIN {X 0,Y 476.03,Z 270.037,A -85,B 0,C 180,E1 -7303.066,E2 -7303.066} C_VEL
LIN {X 0,Y 476.434,Z 259.4,A -85,B 0,C 180,E1 -7303.761,E2 -7303.761} C_VEL
LIN {X 0,Y 476.909,Z 247.759,A -85,B 0,C 180,E1 -7304.345,E2 -7304.345} C_VEL
LIN {X 0,Y 476.929,Z 239.058,A -85,B 0,C 180,E1 -7304.685,E2 -7304.685} C_VEL
LIN {X 0,Y 474.752,Z 226.22,A -85,B 0,C 180,E1 -7305.111,E2 -7305.111} C_VEL
LIN {X 0,Y 474.273,Z 223.447,A -85,B 0,C 180,E1 -7305.195,E2 -7305.195} C_VEL
LIN {X 0,Y 474.551,Z 212.916,A -85,B 0,C 180,E1 -7308.589,E2 -7308.589} C_VEL
LIN {X 0,Y 474.754,Z 203.302,A -85,B 0,C 180,E1 -7311.721,E2 -7311.721} C_VEL
LIN {X 0,Y 475.055,Z 193.62,A -85,B 0,C 180,E1 -7314.938,E2 -7314.938} C_VEL
LIN {X 0,Y 475.434,Z 184.261,A -85,B 0,C 180,E1 -7318.232,E2 -7318.232} C_VEL
LIN {X 0,Y 475.796,Z 174.93,A -85,B 0,C 180,E1 -7321.626,E2 -7321.626} C_VEL
LIN {X 0,Y 476.254,Z 167.102,A -85,B 0,C 180,E1 -7324.647,E2 -7324.647} C_VEL
LIN {X 0,Y 476.325,Z 163.346,A -85,B 0,C 180,E1 -7326.17,E2 -7326.17} C_VEL
LIN {X 0,Y 475.51,Z 158.233,A -85,B 0,C 180,E1 -7328.432,E2 -7328.432} C_VEL
LIN {X 0,Y 474.631,Z 153.366,A -85,B 0,C 180,E1 -7330.808,E2 -7330.808} C_VEL
LIN {X 0,Y 474.614,Z 153.368,A -85,B 0,C 180,E1 -7334.105,E2 -7334.105} C_VEL
LIN {X 0,Y 474.619,Z 153.368,A -85,B 0,C 180,E1 -7337.066,E2 -7337.066} C_VEL
LIN {X 0,Y 474.649,Z 153.365,A -85,B 0,C 180,E1 -7340.454,E2 -7340.454} C_VEL
LIN {X 0,Y 474.593,Z 153.37,A -85,B 0,C 180,E1 -7343.676,E2 -7343.676} C_VEL
LIN {X 0,Y 474.648,Z 153.363,A -85,B 0,C 180,E1 -7346.78,E2 -7346.78} C_VEL
LIN {X 0,Y 474.61,Z 153.368,A -85,B 0,C 180,E1 -7349.77,E2 -7349.77} C_VEL
LIN {X 0,Y 474.702,Z 153.356,A -85,B 0,C 180,E1 -7352.68,E2 -7352.68} C_VEL
LIN {X 0,Y 474.662,Z 153.361,A -85,B 0,C 180,E1 -7355.507,E2 -7355.507} C_VEL
LIN {X 0,Y 474.675,Z 153.36,A -85,B 0,C 180,E1 -7359.185,E2 -7359.185} C_VEL
LIN {X 0,Y 474.651,Z 153.36,A -85,B 0,C 180,E1 -7361.884,E2 -7361.884} C_VEL
LIN {X 0,Y 474.704,Z 153.357,A -85,B 0,C 180,E1 -7364.544,E2 -7364.544} C_VEL
LIN {X 0,Y 474.709,Z 153.355,A -85,B 0,C 180,E1 -7368.037,E2 -7368.037} C_VEL
LIN {X 0,Y 474.733,Z 153.354,A -85,B 0,C 180,E1 -7371.486,E2 -7371.486} C_VEL
LIN {X 0,Y 474.784,Z 153.345,A -85,B 0,C 180,E1 -7374.052,E2 -7374.052} C_VEL
LIN {X 0,Y 474.899,Z 153.332,A -85,B 0,C 180,E1 -7377.455,E2 -7377.455} C_VEL
LIN {X 0,Y 474.917,Z 153.33,A -85,B 0,C 180,E1 -7380,E2 -7380} C_VEL
LIN {X 0,Y 474.898,Z 153.332,A -85,B 0,C 180,E1 -7382.544,E2 -7382.544} C_VEL
LIN {X 0,Y 474.782,Z 153.349,A -85,B 0,C 180,E1 -7385.947,E2 -7385.947} C_VEL
LIN {X 0,Y 474.714,Z 153.357,A -85,B 0,C 180,E1 -7388.513,E2 -7388.513} C_VEL
LIN {X 0,Y 474.438,Z 153.394,A -85,B 0,C 180,E1 -7391.103,E2 -7391.103} C_VEL
LIN {X 0,Y 474.41,Z 154.012,A -85,B 0,C 180,E1 -7392.111,E2 -7392.111} C_VEL
LIN {X 0,Y 474.331,Z 157.698,A -85,B 0,C 180,E1 -7395.616,E2 -7395.616} C_VEL
LIN {X 0,Y 474.175,Z 161.295,A -85,B 0,C 180,E1 -7399.03,E2 -7399.03} C_VEL
LIN {X 0,Y 474.09,Z 164.165,A -85,B 0,C 180,E1 -7401.752,E2 -7401.752} C_VEL
LIN {X 0,Y 474.042,Z 167.136,A -85,B 0,C 180,E1 -7404.526,E2 -7404.526} C_VEL
LIN {X 0,Y 474.037,Z 170.169,A -85,B 0,C 180,E1 -7407.361,E2 -7407.361} C_VEL
LIN {X 0,Y 474.031,Z 172.995,A -85,B 0,C 180,E1 -7409.963,E2 -7409.963} C_VEL
LIN {X 0,Y 477.227,Z 186.848,A -85,B 0,C 180,E1 -7410.506,E2 -7410.506} C_VEL
LIN {X 0,Y 476.9,Z 199.181,A -85,B 0,C 180,E1 -7411.05,E2 -7411.05} C_VEL
LIN {X 0,Y 476.457,Z 210.808,A -85,B 0,C 180,E1 -7411.739,E2 -7411.739} C_VEL
LIN {X 0,Y 476.057,Z 222.182,A -85,B 0,C 180,E1 -7412.604,E2 -7412.604} C_VEL
LIN {X 0,Y 475.658,Z 231.86,A -85,B 0,C 180,E1 -7413.519,E2 -7413.519} C_VEL
LIN {X 0,Y 475.278,Z 240.934,A -85,B 0,C 180,E1 -7414.572,E2 -7414.572} C_VEL
LIN {X 0,Y 474.77,Z 250.027,A -85,B 0,C 180,E1 -7415.879,E2 -7415.879} C_VEL
LIN {X 0,Y 474.499,Z 256.892,A -85,B 0,C 180,E1 -7417.108,E2 -7417.108} C_VEL
LIN {X 0,Y 474.249,Z 263.056,A -85,B 0,C 180,E1 -7418.491,E2 -7418.491} C_VEL
LIN {X 0,Y 474.055,Z 266.97,A -85,B 0,C 180,E1 -7419.604,E2 -7419.604} C_VEL
LIN {X 0,Y 473.892,Z 271.42,A -85,B 0,C 180,E1 -7421.331,E2 -7421.331} C_VEL
LIN {X 0,Y 473.791,Z 274.099,A -85,B 0,C 180,E1 -7423.026,E2 -7423.026} C_VEL
LIN {X 0,Y 473.716,Z 275.104,A -85,B 0,C 180,E1 -7424.592,E2 -7424.592} C_VEL
LIN {X 0,Y 473.723,Z 275,A -85,B 0,C 180,E1 -7425.791,E2 -7425.791} C_VEL
LIN {X 0,Y 473.787,Z 274.098,A -85,B 0,C 180,E1 -7426.972,E2 -7426.972} C_VEL
LIN {X 0,Y 473.811,Z 272.468,A -85,B 0,C 180,E1 -7428.127,E2 -7428.127} C_VEL
LIN {X 0,Y 473.907,Z 270.119,A -85,B 0,C 180,E1 -7429.268,E2 -7429.268} C_VEL
LIN {X 0,Y 474.052,Z 266.898,A -85,B 0,C 180,E1 -7430.436,E2 -7430.436} C_VEL
LIN {X 0,Y 474.23,Z 262.107,A -85,B 0,C 180,E1 -7431.761,E2 -7431.761} C_VEL
LIN {X 0,Y 474.467,Z 255.836,A -85,B 0,C 180,E1 -7433.117,E2 -7433.117} C_VEL
LIN {X 0,Y 474.839,Z 247.819,A -85,B 0,C 180,E1 -7434.492,E2 -7434.492} C_VEL
LIN {X 0,Y 475.274,Z 239.112,A -85,B 0,C 180,E1 -7435.683,E2 -7435.683} C_VEL
LIN {X 0,Y 475.663,Z 229.681,A -85,B 0,C 180,E1 -7436.734,E2 -7436.734} C_VEL
LIN {X 0,Y 476.054,Z 219.032,A -85,B 0,C 180,E1 -7437.697,E2 -7437.697} C_VEL
LIN {X 0,Y 476.435,Z 207.891,A -85,B 0,C 180,E1 -7438.499,E2 -7438.499} C_VEL
LIN {X 0,Y 476.92,Z 196.134,A -85,B 0,C 180,E1 -7439.15,E2 -7439.15} C_VEL
LIN {X 0,Y 477.017,Z 185.704,A -85,B 0,C 180,E1 -7439.598,E2 -7439.598} C_VEL
LIN {X 0,Y 476.664,Z 184.126,A -85,B 0,C 180,E1 -7439.667,E2 -7439.667} C_VEL
LIN {X 0,Y 475.17,Z 180.48,A -85,B 0,C 180,E1 -7439.859,E2 -7439.859} C_VEL
LIN {X 0,Y 472.884,Z 177.405,A -85,B 0,C 180,E1 -7440.095,E2 -7440.095} C_VEL
LIN {X 0,Y 469.639,Z 174.153,A -85,B 0,C 180,E1 -7440.494,E2 -7440.494} C_VEL
LIN {X 0,Y 467.44,Z 172.132,A -85,B 0,C 180,E1 -7440.949,E2 -7440.949} C_VEL
LIN {X 0,Y 466.819,Z 171.308,A -85,B 0,C 180,E1 -7441.338,E2 -7441.338} C_VEL
LIN {X 0,Y 466.903,Z 168.169,A -85,B 0,C 180,E1 -7444.118,E2 -7444.118} C_VEL
LIN {X 0,Y 466.91,Z 164.999,A -85,B 0,C 180,E1 -7446.961,E2 -7446.961} C_VEL
LIN {X 0,Y 466.922,Z 161.936,A -85,B 0,C 180,E1 -7449.745,E2 -7449.745} C_VEL
LIN {X 0,Y 467.02,Z 158.941,A -85,B 0,C 180,E1 -7452.484,E2 -7452.484} C_VEL
LIN {X 0,Y 467.114,Z 156.02,A -85,B 0,C 180,E1 -7455.18,E2 -7455.18} C_VEL
LIN {X 0,Y 467.153,Z 154.299,A -85,B 0,C 180,E1 -7456.958,E2 -7456.958} C_VEL
LIN {X 0,Y 467.485,Z 154.255,A -85,B 0,C 180,E1 -7459.607,E2 -7459.607} C_VEL
LIN {X 0,Y 467.726,Z 154.225,A -85,B 0,C 180,E1 -7462.612,E2 -7462.612} C_VEL
LIN {X 0,Y 467.718,Z 154.226,A -85,B 0,C 180,E1 -7464.827,E2 -7464.827} C_VEL
LIN {X 0,Y 467.857,Z 154.207,A -85,B 0,C 180,E1 -7467.417,E2 -7467.417} C_VEL
LIN {X 0,Y 467.88,Z 154.208,A -85,B 0,C 180,E1 -7470,E2 -7470} C_VEL
LIN {X 0,Y 467.857,Z 154.207,A -85,B 0,C 180,E1 -7472.583,E2 -7472.583} C_VEL
LIN {X 0,Y 467.731,Z 154.225,A -85,B 0,C 180,E1 -7476.037,E2 -7476.037} C_VEL
LIN {X 0,Y 467.678,Z 154.229,A -85,B 0,C 180,E1 -7478.643,E2 -7478.643} C_VEL
LIN {X 0,Y 467.653,Z 154.234,A -85,B 0,C 180,E1 -7482.145,E2 -7482.145} C_VEL
LIN {X 0,Y 467.636,Z 154.238,A -85,B 0,C 180,E1 -7485.695,E2 -7485.695} C_VEL
LIN {X 0,Y 467.614,Z 154.236,A -85,B 0,C 180,E1 -7488.765,E2 -7488.765} C_VEL
LIN {X 0,Y 467.578,Z 154.243,A -85,B 0,C 180,E1 -7491.269,E2 -7491.269} C_VEL
LIN {X 0,Y 467.571,Z 154.245,A -85,B 0,C 180,E1 -7493.943,E2 -7493.943} C_VEL
LIN {X 0,Y 467.613,Z 154.239,A -85,B 0,C 180,E1 -7496.8,E2 -7496.8} C_VEL
LIN {X 0,Y 467.551,Z 154.247,A -85,B 0,C 180,E1 -7499.738,E2 -7499.738} C_VEL
LIN {X 0,Y 467.58,Z 154.243,A -85,B 0,C 180,E1 -7502.759,E2 -7502.759} C_VEL
LIN {X 0,Y 467.55,Z 154.247,A -85,B 0,C 180,E1 -7505.89,E2 -7505.89} C_VEL
LIN {X 0,Y 467.58,Z 154.243,A -85,B 0,C 180,E1 -7509.145,E2 -7509.145} C_VEL
LIN {X 0,Y 467.584,Z 154.243,A -85,B 0,C 180,E1 -7512.567,E2 -7512.567} C_VEL
LIN {X 0,Y 467.568,Z 154.245,A -85,B 0,C 180,E1 -7515.054,E2 -7515.054} C_VEL
LIN {X 0,Y 467.586,Z 154.241,A -85,B 0,C 180,E1 -7517.44,E2 -7517.44} C_VEL
LIN {X 0,Y 467.58,Z 154.244,A -85,B 0,C 180,E1 -7520.856,E2 -7520.856} C_VEL
LIN {X 0,Y 467.56,Z 154.245,A -85,B 0,C 180,E1 -7524.261,E2 -7524.261} C_VEL
LIN {X 0,Y 467.579,Z 154.242,A -85,B 0,C 180,E1 -7527.322,E2 -7527.322} C_VEL
LIN {X 0,Y 467.569,Z 154.245,A -85,B 0,C 180,E1 -7530.668,E2 -7530.668} C_VEL
LIN {X 0,Y 467.616,Z 154.237,A -85,B 0,C 180,E1 -7533.2,E2 -7533.2} C_VEL
LIN {X 0,Y 467.592,Z 154.243,A -85,B 0,C 180,E1 -7536.469,E2 -7536.469} C_VEL
LIN {X 0,Y 467.623,Z 154.236,A -85,B 0,C 180,E1 -7539.778,E2 -7539.778} C_VEL
LIN {X 0,Y 467.598,Z 154.242,A -85,B 0,C 180,E1 -7542.507,E2 -7542.507} C_VEL
LIN {X 0,Y 467.606,Z 154.237,A -85,B 0,C 180,E1 -7545.197,E2 -7545.197} C_VEL
LIN {X 0,Y 467.657,Z 154.233,A -85,B 0,C 180,E1 -7547.855,E2 -7547.855} C_VEL
LIN {X 0,Y 467.672,Z 154.23,A -85,B 0,C 180,E1 -7551.358,E2 -7551.358} C_VEL
LIN {X 0,Y 467.743,Z 154.222,A -85,B 0,C 180,E1 -7553.963,E2 -7553.963} C_VEL
LIN {X 0,Y 467.861,Z 154.207,A -85,B 0,C 180,E1 -7557.418,E2 -7557.418} C_VEL
LIN {X 0,Y 467.885,Z 154.205,A -85,B 0,C 180,E1 -7560,E2 -7560} C_VEL
LIN {X 0,Y 467.861,Z 154.208,A -85,B 0,C 180,E1 -7562.583,E2 -7562.583} C_VEL
LIN {X 0,Y 467.725,Z 154.225,A -85,B 0,C 180,E1 -7566.038,E2 -7566.038} C_VEL
LIN {X 0,Y 467.671,Z 154.231,A -85,B 0,C 180,E1 -7568.643,E2 -7568.643} C_VEL
LIN {X 0,Y 467.658,Z 154.233,A -85,B 0,C 180,E1 -7572.146,E2 -7572.146} C_VEL
LIN {X 0,Y 467.641,Z 154.235,A -85,B 0,C 180,E1 -7575.695,E2 -7575.695} C_VEL
LIN {X 0,Y 467.62,Z 154.237,A -85,B 0,C 180,E1 -7578.765,E2 -7578.765} C_VEL
LIN {X 0,Y 467.583,Z 154.244,A -85,B 0,C 180,E1 -7581.269,E2 -7581.269} C_VEL
LIN {X 0,Y 467.574,Z 154.243,A -85,B 0,C 180,E1 -7583.944,E2 -7583.944} C_VEL
LIN {X 0,Y 467.619,Z 154.236,A -85,B 0,C 180,E1 -7586.801,E2 -7586.801} C_VEL
LIN {X 0,Y 467.556,Z 154.246,A -85,B 0,C 180,E1 -7589.738,E2 -7589.738} C_VEL
LIN {X 0,Y 467.581,Z 154.241,A -85,B 0,C 180,E1 -7592.759,E2 -7592.759} C_VEL
LIN {X 0,Y 467.555,Z 154.244,A -85,B 0,C 180,E1 -7595.89,E2 -7595.89} C_VEL
LIN {X 0,Y 467.578,Z 154.245,A -85,B 0,C 180,E1 -7599.146,E2 -7599.146} C_VEL
LIN {X 0,Y 467.589,Z 154.24,A -85,B 0,C 180,E1 -7602.567,E2 -7602.567} C_VEL
LIN {X 0,Y 467.573,Z 154.24,A -85,B 0,C 180,E1 -7605.053,E2 -7605.053} C_VEL
LIN {X 0,Y 467.591,Z 154.239,A -85,B 0,C 180,E1 -7607.44,E2 -7607.44} C_VEL
LIN {X 0,Y 467.601,Z 154.279,A -85,B 0,C 180,E1 -7609.029,E2 -7609.029} C_VEL
LIN {X 0,Y 468.809,Z 161.018,A -85,B 0,C 180,E1 -7612.074,E2 -7612.074} C_VEL
LIN {X 0,Y 469.382,Z 165.403,A -85,B 0,C 180,E1 -7613.954,E2 -7613.954} C_VEL
LIN {X 0,Y 469.159,Z 171.381,A -85,B 0,C 180,E1 -7616.34,E2 -7616.34} C_VEL
LIN {X 0,Y 468.811,Z 179.235,A -85,B 0,C 180,E1 -7619.356,E2 -7619.356} C_VEL
LIN {X 0,Y 468.347,Z 188.437,A -85,B 0,C 180,E1 -7622.762,E2 -7622.762} C_VEL
LIN {X 0,Y 467.915,Z 197.734,A -85,B 0,C 180,E1 -7626.075,E2 -7626.075} C_VEL
LIN {X 0,Y 467.645,Z 207.352,A -85,B 0,C 180,E1 -7629.319,E2 -7629.319} C_VEL
LIN {X 0,Y 467.4,Z 215.55,A -85,B 0,C 180,E1 -7632.047,E2 -7632.047} C_VEL
LIN {X 0,Y 467.25,Z 223.203,A -85,B 0,C 180,E1 -7634.571,E2 -7634.571} C_VEL
LIN {X 0,Y 469.833,Z 238.753,A -85,B 0,C 180,E1 -7635.088,E2 -7635.088} C_VEL
LIN {X 0,Y 470.138,Z 243.588,A -85,B 0,C 180,E1 -7635.278,E2 -7635.278} C_VEL
LIN {X 0,Y 469.742,Z 255.256,A -85,B 0,C 180,E1 -7635.819,E2 -7635.819} C_VEL
LIN {X 0,Y 469.273,Z 266.483,A -85,B 0,C 180,E1 -7636.5,E2 -7636.5} C_VEL
LIN {X 0,Y 468.844,Z 276.995,A -85,B 0,C 180,E1 -7637.306,E2 -7637.306} C_VEL
LIN {X 0,Y 468.383,Z 287.597,A -85,B 0,C 180,E1 -7638.313,E2 -7638.313} C_VEL
LIN {X 0,Y 467.876,Z 296.786,A -85,B 0,C 180,E1 -7639.397,E2 -7639.397} C_VEL
LIN {X 0,Y 467.447,Z 305.688,A -85,B 0,C 180,E1 -7640.699,E2 -7640.699} C_VEL
LIN {X 0,Y 467.093,Z 312.849,A -85,B 0,C 180,E1 -7642,E2 -7642} C_VEL
LIN {X 0,Y 466.904,Z 319.091,A -85,B 0,C 180,E1 -7643.444,E2 -7643.444} C_VEL
LIN {X 0,Y 466.784,Z 323.677,A -85,B 0,C 180,E1 -7644.817,E2 -7644.817} C_VEL
LIN {X 0,Y 466.663,Z 325.958,A -85,B 0,C 180,E1 -7645.682,E2 -7645.682} C_VEL
LIN {X 0,Y 466.695,Z 327.807,A -85,B 0,C 180,E1 -7646.547,E2 -7646.547} C_VEL
LIN {X 0,Y 466.647,Z 329.193,A -85,B 0,C 180,E1 -7647.411,E2 -7647.411} C_VEL
LIN {X 0,Y 466.59,Z 330.785,A -85,B 0,C 180,E1 -7649.137,E2 -7649.137} C_VEL
LIN {X 0,Y 466.57,Z 331,A -85,B 0,C 180,E1 -7650,E2 -7650} C_VEL
LIN {X 0,Y 466.59,Z 330.786,A -85,B 0,C 180,E1 -7650.863,E2 -7650.863} C_VEL
LIN {X 0,Y 466.647,Z 329.195,A -85,B 0,C 180,E1 -7652.59,E2 -7652.59} C_VEL
LIN {X 0,Y 466.695,Z 327.81,A -85,B 0,C 180,E1 -7653.454,E2 -7653.454} C_VEL
LIN {X 0,Y 466.703,Z 324.895,A -85,B 0,C 180,E1 -7654.751,E2 -7654.751} C_VEL
LIN {X 0,Y 466.841,Z 320.947,A -85,B 0,C 180,E1 -7656.049,E2 -7656.049} C_VEL
LIN {X 0,Y 466.999,Z 314.874,A -85,B 0,C 180,E1 -7657.567,E2 -7657.567} C_VEL
LIN {X 0,Y 467.351,Z 308.234,A -85,B 0,C 180,E1 -7658.867,E2 -7658.867} C_VEL
LIN {X 0,Y 467.74,Z 299.991,A -85,B 0,C 180,E1 -7660.169,E2 -7660.169} C_VEL
LIN {X 0,Y 468.128,Z 291.516,A -85,B 0,C 180,E1 -7661.255,E2 -7661.255} C_VEL
LIN {X 0,Y 468.66,Z 281.186,A -85,B 0,C 180,E1 -7662.32,E2 -7662.32} C_VEL
LIN {X 0,Y 469.093,Z 269.546,A -85,B 0,C 180,E1 -7663.285,E2 -7663.285} C_VEL
LIN {X 0,Y 469.63,Z 257.203,A -85,B 0,C 180,E1 -7664.075,E2 -7664.075} C_VEL
LIN {X 0,Y 470.103,Z 244.826,A -85,B 0,C 180,E1 -7664.668,E2 -7664.668} C_VEL
LIN {X 0,Y 469.969,Z 239.834,A -85,B 0,C 180,E1 -7664.866,E2 -7664.866} C_VEL
LIN {X 0,Y 467.861,Z 227.124,A -85,B 0,C 180,E1 -7665.307,E2 -7665.307} C_VEL
LIN {X 0,Y 467.213,Z 223.103,A -85,B 0,C 180,E1 -7665.43,E2 -7665.43} C_VEL
LIN {X 0,Y 467.485,Z 213.066,A -85,B 0,C 180,E1 -7668.715,E2 -7668.715} C_VEL
LIN {X 0,Y 467.677,Z 204.248,A -85,B 0,C 180,E1 -7671.631,E2 -7671.631} C_VEL
LIN {X 0,Y 467.991,Z 194.701,A -85,B 0,C 180,E1 -7674.866,E2 -7674.866} C_VEL
LIN {X 0,Y 468.403,Z 185.275,A -85,B 0,C 180,E1 -7678.206,E2 -7678.206} C_VEL
LIN {X 0,Y 468.787,Z 176.064,A -85,B 0,C 180,E1 -7681.649,E2 -7681.649} C_VEL
LIN {X 0,Y 469.265,Z 168.313,A -85,B 0,C 180,E1 -7684.689,E2 -7684.689} C_VEL
LIN {X 0,Y 469.374,Z 165.024,A -85,B 0,C 180,E1 -7686.045,E2 -7686.045} C_VEL
LIN {X 0,Y 468.788,Z 160.79,A -85,B 0,C 180,E1 -7687.928,E2 -7687.928} C_VEL
LIN {X 0,Y 467.603,Z 154.242,A -85,B 0,C 180,E1 -7691.112,E2 -7691.112} C_VEL
LIN {X 0,Y 467.559,Z 154.246,A -85,B 0,C 180,E1 -7693.821,E2 -7693.821} C_VEL
LIN {X 0,Y 467.561,Z 154.249,A -85,B 0,C 180,E1 -7696.256,E2 -7696.256} C_VEL
LIN {X 0,Y 467.583,Z 154.246,A -85,B 0,C 180,E1 -7698.723,E2 -7698.723} C_VEL
LIN {X 0,Y 467.569,Z 154.247,A -85,B 0,C 180,E1 -7701.955,E2 -7701.955} C_VEL
LIN {X 0,Y 467.569,Z 154.246,A -85,B 0,C 180,E1 -7705.167,E2 -7705.167} C_VEL
LIN {X 0,Y 467.588,Z 154.243,A -85,B 0,C 180,E1 -7708.26,E2 -7708.26} C_VEL
LIN {X 0,Y 467.582,Z 154.242,A -85,B 0,C 180,E1 -7711.25,E2 -7711.25} C_VEL
LIN {X 0,Y 467.621,Z 154.237,A -85,B 0,C 180,E1 -7713.2,E2 -7713.2} C_VEL
LIN {X 0,Y 467.597,Z 154.243,A -85,B 0,C 180,E1 -7716.468,E2 -7716.468} C_VEL
LIN {X 0,Y 467.627,Z 154.236,A -85,B 0,C 180,E1 -7719.777,E2 -7719.777} C_VEL
LIN {X 0,Y 467.603,Z 154.24,A -85,B 0,C 180,E1 -7722.506,E2 -7722.506} C_VEL
